KUKA KRL program: f1_Kuka_APT203T02S03.SRC

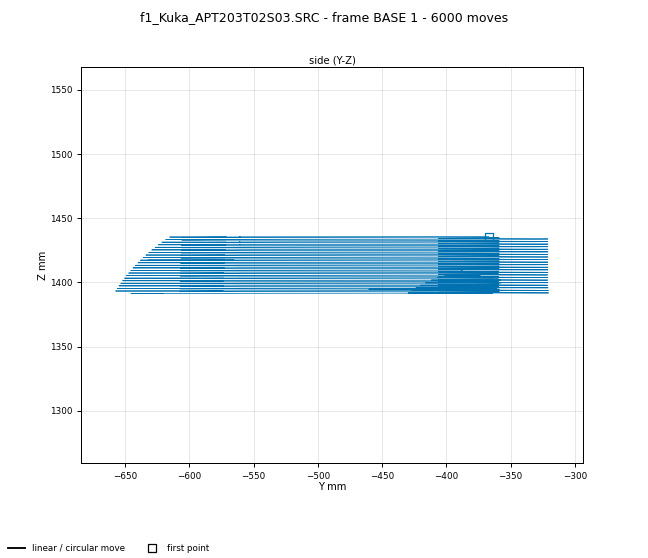
[picture p0: tool path of f1_Kuka_APT203T02S03.SRC in frame BASE 1, 6000 of 6001 moves have a stored position in this frame; points joined in program order, loops and branches not executed]
&ACCESS RVP
&REL 2
&PARAM TEMPLATE = C:\KRC\Roboter\Template\vorgabe
&PARAM EDITMASK = *
DEF f1_Kuka_APT203T02S03()


;FOLD INI;%{PE}%V3.2.0,%MKUKATPBASIS,%CINIT,%VCOMMON,%P
  ;FOLD BAS INI;%{E}%V3.2.0,%MKUKATPBASIS,%CINIT,%VINIT,%P
    GLOBAL INTERRUPT DECL 3 WHEN $STOPMESS==TRUE DO IR_STOPM ( )
    INTERRUPT ON 3
    BAS (#INITMOV,0 )
  ;ENDFOLD (BAS INI)
  ;FOLD USER INI;%{E}%V3.2.0,%MKUKATPUSER,%CINIT,%VINIT,%P
    ;Make your modifications here
  ;ENDFOLD (USER INI)
;ENDFOLD (INI)


;*** Make Null PTP Move
  PTP $pos_act

;*** Auto Load The Correct TOOL Data
  $tool=tool_data[2]

;*** Auto Load The Correct BASE Data
  $base=base_data[1]

  $ADVANCE = 5

;*** Restate Last Velocity
MMPM(30000.0)
SetRPM(8000)
LIN {X 0.139,Y -366.989,Z 1435.725,A 0.000,B 0.000,C 90.000,E1 166.408} C_DIS
LIN {X -0.133,Y -369.731,Z 1435.724,A 0.000,B 0.000,C 90.000,E1 166.284} C_DIS
LIN {X -0.049,Y -372.656,Z 1435.723,A 0.000,B 0.000,C 90.000,E1 166.061} C_DIS
LIN {X -0.133,Y -378.778,Z 1435.720,A 0.000,B 0.000,C 90.000,E1 165.574} C_DIS
LIN {X -0.061,Y -386.543,Z 1435.716,A 0.000,B 0.000,C 90.000,E1 164.866} C_DIS
LIN {X 0.126,Y -394.122,Z 1435.712,A 0.000,B 0.000,C 90.000,E1 164.102} C_DIS
LIN {X -0.061,Y -412.834,Z 1435.702,A 0.000,B 0.000,C 90.000,E1 162.417} C_DIS
LIN {X -0.188,Y -426.811,Z 1435.696,A 0.000,B 0.000,C 90.000,E1 161.221} C_DIS
LIN {X 0.041,Y -439.162,Z 1435.690,A 0.000,B 0.000,C 90.000,E1 160.134} C_DIS
LIN {X -0.042,Y -454.601,Z 1435.682,A 0.000,B 0.000,C 90.000,E1 158.847} C_DIS
LIN {X -0.244,Y -463.730,Z 1435.678,A 0.000,B 0.000,C 90.000,E1 158.103} C_DIS
LIN {X -0.043,Y -474.282,Z 1435.673,A 0.000,B 0.000,C 90.000,E1 157.177} C_DIS
LIN {X 0.193,Y -484.648,Z 1435.668,A 0.000,B 0.000,C 90.000,E1 156.230} C_DIS
LIN {X 0.112,Y -493.177,Z 1435.664,A 0.000,B 0.000,C 90.000,E1 155.433} C_DIS
LIN {X -0.238,Y -500.193,Z 1435.660,A 0.000,B 0.000,C 90.000,E1 154.793} C_DIS
LIN {X -0.084,Y -506.867,Z 1435.656,A 0.000,B 0.000,C 90.000,E1 154.076} C_DIS
LIN {X -0.024,Y -510.765,Z 1435.654,A 0.000,B 0.000,C 90.000,E1 153.640} C_DIS
LIN {X -0.152,Y -516.626,Z 1435.650,A 0.000,B 0.000,C 90.000,E1 152.922} C_DIS
LIN {X -0.204,Y -519.973,Z 1435.647,A 0.000,B 0.000,C 90.000,E1 152.487} C_DIS
LIN {X -0.159,Y -524.000,Z 1435.644,A 0.000,B 0.000,C 90.000,E1 151.897} C_DIS
LIN {X -0.081,Y -527.512,Z 1435.641,A 0.000,B 0.000,C 90.000,E1 151.307} C_DIS
LIN {X -0.125,Y -531.403,Z 1435.637,A 0.000,B 0.000,C 90.000,E1 150.589} C_DIS
LIN {X 0.009,Y -534.231,Z 1435.633,A 0.000,B 0.000,C 90.000,E1 149.999} C_DIS
LIN {X 0.019,Y -537.257,Z 1435.629,A 0.000,B 0.000,C 90.000,E1 149.282} C_DIS
LIN {X -0.271,Y -539.517,Z 1435.626,A 0.000,B 0.000,C 90.000,E1 148.742} C_DIS
LIN {X -0.078,Y -542.313,Z 1435.621,A 0.000,B 0.000,C 90.000,E1 147.867} C_DIS
LIN {X -0.041,Y -544.044,Z 1435.618,A 0.000,B 0.000,C 90.000,E1 147.296} C_DIS
LIN {X -0.062,Y -547.087,Z 1435.612,A 0.000,B 0.000,C 90.000,E1 146.167} C_DIS
LIN {X 0.115,Y -549.696,Z 1435.606,A 0.000,B 0.000,C 90.000,E1 145.022} C_DIS
LIN {X -0.096,Y -550.840,Z 1435.603,A 0.000,B 0.000,C 90.000,E1 144.482} C_DIS
LIN {X 0.145,Y -552.809,Z 1435.596,A 0.000,B 0.000,C 90.000,E1 143.336} C_DIS
LIN {X 0.346,Y -554.026,Z 1435.592,A 0.000,B 0.000,C 90.000,E1 142.477} C_DIS
LIN {X 0.271,Y -555.675,Z 1435.584,A 0.000,B 0.000,C 90.000,E1 141.090} C_DIS
LIN {X 0.141,Y -556.707,Z 1435.578,A 0.000,B 0.000,C 90.000,E1 139.989} C_DIS
LIN {X 0.039,Y -557.845,Z 1435.570,A 0.000,B 0.000,C 90.000,E1 138.609} C_DIS
LIN {X -0.041,Y -558.827,Z 1435.562,A 0.000,B 0.000,C 90.000,E1 137.229} C_DIS
LIN {X -0.185,Y -559.579,Z 1435.556,A 0.000,B 0.000,C 90.000,E1 136.134} C_DIS
LIN {X 0.071,Y -560.088,Z 1435.550,A 0.000,B 0.000,C 90.000,E1 135.000} C_DIS
LIN {X 0.002,Y -560.630,Z 1435.542,A 0.000,B 0.000,C 90.000,E1 133.623} C_DIS
LIN {X -0.035,Y -560.945,Z 1435.535,A 0.000,B 0.000,C 90.000,E1 132.243} C_DIS
LIN {X -0.060,Y -561.072,Z 1435.527,A 0.000,B 0.000,C 90.000,E1 130.862} C_DIS
LIN {X 0.097,Y -561.162,Z 1435.516,A 0.000,B 0.000,C 90.000,E1 128.910} C_DIS
LIN {X 0.142,Y -561.163,Z 1435.509,A 0.000,B 0.000,C 90.000,E1 127.523} C_DIS
LIN {X -0.055,Y -561.053,Z 1435.499,A 0.000,B 0.000,C 90.000,E1 125.884} C_DIS
LIN {X 0.103,Y -560.922,Z 1435.492,A 0.000,B 0.000,C 90.000,E1 124.485} C_DIS
LIN {X 0.254,Y -560.635,Z 1435.484,A 0.000,B 0.000,C 90.000,E1 123.086} C_DIS
LIN {X 0.083,Y -560.385,Z 1435.476,A 0.000,B 0.000,C 90.000,E1 121.720} C_DIS
LIN {X -0.090,Y -560.625,Z 1435.459,A 0.000,B 0.000,C 90.000,E1 118.693} C_DIS
LIN {X 0.023,Y -561.190,Z 1435.449,A 0.000,B 0.000,C 90.000,E1 116.744} C_DIS
LIN {X 0.086,Y -561.848,Z 1435.439,A 0.000,B 0.000,C 90.000,E1 115.079} C_DIS
LIN {X 0.115,Y -562.232,Z 1435.432,A 0.000,B 0.000,C 90.000,E1 113.695} C_DIS
LIN {X 0.247,Y -562.726,Z 1435.423,A 0.000,B 0.000,C 90.000,E1 112.025} C_DIS
LIN {X 0.174,Y -563.696,Z 1435.416,A 0.000,B 0.000,C 90.000,E1 110.791} C_DIS
LIN {X 0.095,Y -564.430,Z 1435.414,A 0.000,B 0.000,C 90.000,E1 110.482} C_DIS
LIN {X -0.307,Y -564.927,Z 1435.412,A 0.000,B 0.000,C 90.000,E1 110.248} C_DIS
LIN {X -0.215,Y -566.966,Z 1435.411,A 0.000,B 0.000,C 90.000,E1 109.939} C_DIS
LIN {X 0.217,Y -568.542,Z 1435.410,A 0.000,B 0.000,C 90.000,E1 109.758} C_DIS
LIN {X -0.209,Y -571.322,Z 1435.409,A 0.000,B 0.000,C 90.000,E1 109.577} C_DIS
LIN {X -0.175,Y -580.313,Z 1435.406,A 0.000,B 0.000,C 90.000,E1 109.014} C_DIS
LIN {X 0.231,Y -583.140,Z 1435.405,A 0.000,B 0.000,C 90.000,E1 108.779} C_DIS
LIN {X -0.178,Y -587.504,Z 1435.403,A 0.000,B 0.000,C 90.000,E1 108.489} C_DIS
LIN {X 0.008,Y -592.694,Z 1435.400,A 0.000,B 0.000,C 90.000,E1 108.000} C_DIS
LIN {X 0.320,Y -597.592,Z 1435.397,A 0.000,B 0.000,C 90.000,E1 107.457} C_DIS
LIN {X -0.290,Y -602.793,Z 1435.394,A 0.000,B 0.000,C 90.000,E1 106.858} C_DIS
LIN {X -0.042,Y -605.424,Z 1435.391,A 0.000,B 0.000,C 90.000,E1 106.441} C_DIS
LIN {X -0.313,Y -607.026,Z 1435.390,A 0.000,B 0.000,C 90.000,E1 106.205} C_DIS
LIN {X -0.042,Y -608.899,Z 1435.388,A 0.000,B 0.000,C 90.000,E1 105.788} C_DIS
LIN {X 0.194,Y -610.823,Z 1435.385,A 0.000,B 0.000,C 90.000,E1 105.245} C_DIS
LIN {X -0.060,Y -611.515,Z 1435.383,A 0.000,B 0.000,C 90.000,E1 105.009} C_DIS
LIN {X 0.034,Y -612.594,Z 1435.380,A 0.000,B 0.000,C 90.000,E1 104.481} C_DIS
LIN {X 0.042,Y -613.900,Z 1435.376,A 0.000,B 0.000,C 90.000,E1 103.703} C_DIS
LIN {X -0.086,Y -614.813,Z 1435.372,A 0.000,B 0.000,C 90.000,E1 102.939} C_DIS
LIN {X 0.033,Y -615.205,Z 1435.369,A 0.000,B 0.000,C 90.000,E1 102.411} C_DIS
LIN {X 0.156,Y -615.334,Z 1435.366,A 0.000,B 0.000,C 90.000,E1 101.883} C_DIS
LIN {X 0.158,Y -615.193,Z 1435.363,A 0.000,B 0.000,C 90.000,E1 101.366} C_DIS
LIN {X 0.283,Y -614.654,Z 1435.360,A 0.000,B 0.000,C 90.000,E1 100.838} C_DIS
LIN {X -0.202,Y -613.771,Z 1435.358,A 0.000,B 0.000,C 90.000,E1 100.366} C_DIS
LIN {X -0.197,Y -612.563,Z 1435.355,A 0.000,B 0.000,C 90.000,E1 99.849} C_DIS
LIN {X -0.095,Y -611.088,Z 1435.352,A 0.000,B 0.000,C 90.000,E1 99.321} C_DIS
LIN {X 0.252,Y -610.301,Z 1435.350,A 0.000,B 0.000,C 90.000,E1 99.029} C_DIS
LIN {X 0.239,Y -608.456,Z 1435.347,A 0.000,B 0.000,C 90.000,E1 98.511} C_DIS
LIN {X 0.123,Y -605.414,Z 1435.344,A 0.000,B 0.000,C 90.000,E1 97.871} C_DIS
LIN {X 0.016,Y -599.697,Z 1435.338,A 0.000,B 0.000,C 90.000,E1 96.834} C_DIS
LIN {X -0.252,Y -595.611,Z 1435.334,A 0.000,B 0.000,C 90.000,E1 96.201} C_DIS
LIN {X 0.231,Y -591.760,Z 1435.331,A 0.000,B 0.000,C 90.000,E1 95.625} C_DIS
LIN {X 0.011,Y -585.389,Z 1435.328,A 0.000,B 0.000,C 90.000,E1 94.992} C_DIS
LIN {X -0.058,Y -578.085,Z 1435.325,A 0.000,B 0.000,C 90.000,E1 94.416} C_DIS
LIN {X 0.163,Y -573.369,Z 1435.322,A 0.000,B 0.000,C 90.000,E1 93.955} C_DIS
LIN {X -0.164,Y -571.760,Z 1435.320,A 0.000,B 0.000,C 90.000,E1 93.669} C_DIS
LIN {X -0.139,Y -571.146,Z 1435.318,A 0.000,B 0.000,C 90.000,E1 93.326} C_DIS
LIN {X 0.212,Y -571.043,Z 1435.318,A 0.000,B 0.000,C 90.000,E1 93.154} C_DIS
LIN {X 0.110,Y -571.148,Z 1435.313,A 0.000,B 0.000,C 90.000,E1 92.350} C_DIS
LIN {X -0.222,Y -573.341,Z 1435.298,A 0.000,B 0.000,C 90.000,E1 89.656} C_DIS
LIN {X -0.082,Y -574.625,Z 1435.290,A 0.000,B 0.000,C 90.000,E1 88.282} C_DIS
LIN {X 0.272,Y -576.117,Z 1435.281,A 0.000,B 0.000,C 90.000,E1 86.617} C_DIS
LIN {X -0.248,Y -577.119,Z 1435.275,A 0.000,B 0.000,C 90.000,E1 85.584} C_DIS
LIN {X 0.219,Y -578.736,Z 1435.266,A 0.000,B 0.000,C 90.000,E1 83.913} C_DIS
LIN {X 0.154,Y -581.189,Z 1435.253,A 0.000,B 0.000,C 90.000,E1 81.489} C_DIS
LIN {X 0.060,Y -582.537,Z 1435.245,A 0.000,B 0.000,C 90.000,E1 80.151} C_DIS
LIN {X 0.141,Y -584.830,Z 1435.233,A 0.000,B 0.000,C 90.000,E1 77.993} C_DIS
LIN {X 0.221,Y -585.974,Z 1435.226,A 0.000,B 0.000,C 90.000,E1 76.645} C_DIS
LIN {X -0.109,Y -586.981,Z 1435.219,A 0.000,B 0.000,C 90.000,E1 75.338} C_DIS
LIN {X -0.098,Y -587.692,Z 1435.213,A 0.000,B 0.000,C 90.000,E1 74.267} C_DIS
LIN {X -0.158,Y -588.617,Z 1435.204,A 0.000,B 0.000,C 90.000,E1 72.670} C_DIS
LIN {X 0.139,Y -589.465,Z 1435.195,A 0.000,B 0.000,C 90.000,E1 71.040} C_DIS
LIN {X 0.101,Y -590.311,Z 1435.186,A 0.000,B 0.000,C 90.000,E1 69.444} C_DIS
LIN {X -0.020,Y -591.408,Z 1435.176,A 0.000,B 0.000,C 90.000,E1 67.592} C_DIS
LIN {X -0.027,Y -592.306,Z 1435.167,A 0.000,B 0.000,C 90.000,E1 65.997} C_DIS
LIN {X -0.274,Y -593.812,Z 1435.155,A 0.000,B 0.000,C 90.000,E1 63.896} C_DIS
LIN {X 0.065,Y -594.884,Z 1435.147,A 0.000,B 0.000,C 90.000,E1 62.538} C_DIS
LIN {X 0.275,Y -597.024,Z 1435.133,A 0.000,B 0.000,C 90.000,E1 59.871} C_DIS
LIN {X -0.248,Y -598.685,Z 1435.123,A 0.000,B 0.000,C 90.000,E1 58.074} C_DIS
LIN {X 0.263,Y -599.902,Z 1435.115,A 0.000,B 0.000,C 90.000,E1 56.707} C_DIS
LIN {X -0.047,Y -601.554,Z 1435.105,A 0.000,B 0.000,C 90.000,E1 54.895} C_DIS
LIN {X -0.219,Y -602.822,Z 1435.096,A 0.000,B 0.000,C 90.000,E1 53.336} C_DIS
LIN {X 0.215,Y -603.813,Z 1435.089,A 0.000,B 0.000,C 90.000,E1 51.984} C_DIS
LIN {X -0.030,Y -604.760,Z 1435.080,A 0.000,B 0.000,C 90.000,E1 50.436} C_DIS
LIN {X -0.183,Y -605.178,Z 1435.076,A 0.000,B 0.000,C 90.000,E1 49.666} C_DIS
LIN {X 0.188,Y -605.443,Z 1435.069,A 0.000,B 0.000,C 90.000,E1 48.324} C_DIS
LIN {X -0.292,Y -605.672,Z 1435.058,A 0.000,B 0.000,C 90.000,E1 46.539} C_DIS
LIN {X 0.030,Y -605.750,Z 1435.051,A 0.000,B 0.000,C 90.000,E1 45.202} C_DIS
LIN {X -0.313,Y -605.439,Z 1435.045,A 0.000,B 0.000,C 90.000,E1 44.190} C_DIS
LIN {X 0.010,Y -604.840,Z 1435.038,A 0.000,B 0.000,C 90.000,E1 42.852} C_DIS
LIN {X -0.085,Y -603.901,Z 1435.031,A 0.000,B 0.000,C 90.000,E1 41.553} C_DIS
LIN {X -0.238,Y -603.180,Z 1435.026,A 0.000,B 0.000,C 90.000,E1 40.782} C_DIS
LIN {X 0.098,Y -601.757,Z 1435.019,A 0.000,B 0.000,C 90.000,E1 39.439} C_DIS
LIN {X 0.157,Y -600.481,Z 1435.013,A 0.000,B 0.000,C 90.000,E1 38.382} C_DIS
LIN {X 0.058,Y -598.543,Z 1435.006,A 0.000,B 0.000,C 90.000,E1 37.076} C_DIS
LIN {X 0.052,Y -596.081,Z 1434.999,A 0.000,B 0.000,C 90.000,E1 35.758} C_DIS
LIN {X -0.136,Y -593.171,Z 1434.991,A 0.000,B 0.000,C 90.000,E1 34.452} C_DIS
LIN {X 0.170,Y -591.220,Z 1434.987,A 0.000,B 0.000,C 90.000,E1 33.627} C_DIS
LIN {X 0.332,Y -588.313,Z 1434.981,A 0.000,B 0.000,C 90.000,E1 32.546} C_DIS
LIN {X -0.097,Y -586.776,Z 1434.978,A 0.000,B 0.000,C 90.000,E1 32.054} C_DIS
LIN {X -0.171,Y -584.094,Z 1434.974,A 0.000,B 0.000,C 90.000,E1 31.258} C_DIS
LIN {X -0.133,Y -582.079,Z 1434.971,A 0.000,B 0.000,C 90.000,E1 30.718} C_DIS
LIN {X -0.112,Y -579.882,Z 1434.968,A 0.000,B 0.000,C 90.000,E1 30.178} C_DIS
LIN {X 0.246,Y -576.285,Z 1434.963,A 0.000,B 0.000,C 90.000,E1 29.333} C_DIS
LIN {X -0.138,Y -572.981,Z 1434.959,A 0.000,B 0.000,C 90.000,E1 28.693} C_DIS
LIN {X 0.146,Y -568.644,Z 1434.955,A 0.000,B 0.000,C 90.000,E1 27.847} C_DIS
LIN {X 0.283,Y -563.075,Z 1434.949,A 0.000,B 0.000,C 90.000,E1 26.873} C_DIS
LIN {X -0.005,Y -556.116,Z 1434.943,A 0.000,B 0.000,C 90.000,E1 25.796} C_DIS
LIN {X 0.079,Y -550.567,Z 1434.939,A 0.000,B 0.000,C 90.000,E1 24.951} C_DIS
LIN {X 0.109,Y -546.505,Z 1434.936,A 0.000,B 0.000,C 90.000,E1 24.387} C_DIS
LIN {X -0.019,Y -540.965,Z 1434.932,A 0.000,B 0.000,C 90.000,E1 23.695} C_DIS
LIN {X 0.300,Y -535.092,Z 1434.928,A 0.000,B 0.000,C 90.000,E1 22.950} C_DIS
LIN {X -0.249,Y -527.574,Z 1434.923,A 0.000,B 0.000,C 90.000,E1 22.153} C_DIS
LIN {X -0.192,Y -518.481,Z 1434.917,A 0.000,B 0.000,C 90.000,E1 21.153} C_DIS
LIN {X -0.220,Y -512.109,Z 1434.914,A 0.000,B 0.000,C 90.000,E1 20.482} C_DIS
LIN {X 0.092,Y -501.330,Z 1434.907,A 0.000,B 0.000,C 90.000,E1 19.322} C_DIS
LIN {X -0.015,Y -487.754,Z 1434.900,A 0.000,B 0.000,C 90.000,E1 17.946} C_DIS
LIN {X -0.074,Y -470.249,Z 1434.889,A 0.000,B 0.000,C 90.000,E1 16.079} C_DIS
LIN {X -0.198,Y -452.851,Z 1434.878,A 0.000,B 0.000,C 90.000,E1 14.120} C_DIS
LIN {X 0.206,Y -444.598,Z 1434.873,A 0.000,B 0.000,C 90.000,E1 13.119} C_DIS
LIN {X -0.161,Y -440.352,Z 1434.870,A 0.000,B 0.000,C 90.000,E1 12.703} C_DIS
LIN {X -0.110,Y -435.815,Z 1434.868,A 0.000,B 0.000,C 90.000,E1 12.243} C_DIS
LIN {X -0.151,Y -431.034,Z 1434.866,A 0.000,B 0.000,C 90.000,E1 11.827} C_DIS
LIN {X 0.079,Y -427.565,Z 1434.864,A 0.000,B 0.000,C 90.000,E1 11.535} C_DIS
LIN {X 0.097,Y -423.730,Z 1434.863,A 0.000,B 0.000,C 90.000,E1 11.299} C_DIS
LIN {X 0.019,Y -420.614,Z 1434.862,A 0.000,B 0.000,C 90.000,E1 11.186} C_DIS
LIN {X -0.096,Y -419.777,Z 1434.862,A 0.000,B 0.000,C 90.000,E1 11.186} C_DIS
LIN {X -0.117,Y -367.196,Z 1434.862,A 0.000,B 0.000,C 90.000,E1 11.186} C_DIS
LIN {X -0.112,Y -366.497,Z 1434.855,A 0.000,B 0.000,C 90.000,E1 9.962} C_DIS
LIN {X 0.185,Y -361.797,Z 1434.822,A 0.000,B 0.000,C 90.000,E1 3.955} C_DIS
LIN {X 0.070,Y -360.903,Z 1434.801,A 0.000,B 0.000,C 90.000,E1 0.229} C_DIS
LIN {X -0.053,Y -359.426,Z 1434.770,A 0.000,B 0.000,C 90.000,E1 354.546} C_DIS
LIN {X 0.070,Y -358.890,Z 1434.759,A 0.000,B 0.000,C 90.000,E1 352.648} C_DIS
LIN {X -0.020,Y -359.563,Z 1434.726,A 0.000,B 0.000,C 90.000,E1 346.645} C_DIS
LIN {X 0.001,Y -361.801,Z 1434.684,A 0.000,B 0.000,C 90.000,E1 339.135} C_DIS
LIN {X -0.154,Y -362.053,Z 1434.680,A 0.000,B 0.000,C 90.000,E1 338.411} C_DIS
LIN {X 0.189,Y -365.980,Z 1434.643,A 0.000,B 0.000,C 90.000,E1 331.641} C_DIS
LIN {X 0.029,Y -366.387,Z 1434.639,A 0.000,B 0.000,C 90.000,E1 330.923} C_DIS
LIN {X -0.031,Y -371.355,Z 1434.604,A 0.000,B 0.000,C 90.000,E1 324.642} C_DIS
LIN {X -0.043,Y -371.766,Z 1434.602,A 0.000,B 0.000,C 90.000,E1 324.276} C_DIS
LIN {X 0.013,Y -377.358,Z 1434.567,A 0.000,B 0.000,C 90.000,E1 318.038} C_DIS
LIN {X 0.012,Y -378.235,Z 1434.563,A 0.000,B 0.000,C 90.000,E1 317.310} C_DIS
LIN {X 0.002,Y -383.940,Z 1434.531,A 0.000,B 0.000,C 90.000,E1 311.515} C_DIS
LIN {X 0.088,Y -384.893,Z 1434.527,A 0.000,B 0.000,C 90.000,E1 310.782} C_DIS
LIN {X 0.262,Y -390.610,Z 1434.495,A 0.000,B 0.000,C 90.000,E1 305.025} C_DIS
LIN {X 0.106,Y -391.104,Z 1434.493,A 0.000,B 0.000,C 90.000,E1 304.692} C_DIS
LIN {X 0.022,Y -391.648,Z 1434.489,A 0.000,B 0.000,C 90.000,E1 303.992} C_DIS
LIN {X -0.080,Y -396.825,Z 1434.459,A 0.000,B 0.000,C 90.000,E1 298.693} C_DIS
LIN {X -0.210,Y -397.120,Z 1434.457,A 0.000,B 0.000,C 90.000,E1 298.359} C_DIS
LIN {X -0.055,Y -401.597,Z 1434.426,A 0.000,B 0.000,C 90.000,E1 292.717} C_DIS
LIN {X 0.222,Y -404.659,Z 1434.395,A 0.000,B 0.000,C 90.000,E1 287.094} C_DIS
LIN {X -0.079,Y -404.735,Z 1434.391,A 0.000,B 0.000,C 90.000,E1 286.441} C_DIS
LIN {X 0.214,Y -406.099,Z 1434.364,A 0.000,B 0.000,C 90.000,E1 281.535} C_DIS
LIN {X -0.176,Y -406.094,Z 1434.362,A 0.000,B 0.000,C 90.000,E1 281.243} C_DIS
LIN {X -0.097,Y -405.680,Z 1434.333,A 0.000,B 0.000,C 90.000,E1 276.024} C_DIS
LIN {X -0.165,Y -405.058,Z 1434.328,A 0.000,B 0.000,C 90.000,E1 274.992} C_DIS
LIN {X -0.060,Y -403.497,Z 1434.304,A 0.000,B 0.000,C 90.000,E1 270.802} C_DIS
LIN {X -0.092,Y -403.288,Z 1434.302,A 0.000,B 0.000,C 90.000,E1 270.458} C_DIS
LIN {X 0.091,Y -398.931,Z 1434.271,A 0.000,B 0.000,C 90.000,E1 264.837} C_DIS
LIN {X -0.040,Y -393.108,Z 1434.242,A 0.000,B 0.000,C 90.000,E1 259.567} C_DIS
LIN {X -0.079,Y -392.835,Z 1434.240,A 0.000,B 0.000,C 90.000,E1 259.218} C_DIS
LIN {X 0.034,Y -385.993,Z 1434.212,A 0.000,B 0.000,C 90.000,E1 254.212} C_DIS
LIN {X -0.026,Y -385.267,Z 1434.208,A 0.000,B 0.000,C 90.000,E1 253.504} C_DIS
LIN {X -0.004,Y -384.768,Z 1434.206,A 0.000,B 0.000,C 90.000,E1 253.142} C_DIS
LIN {X 0.221,Y -377.973,Z 1434.182,A 0.000,B 0.000,C 90.000,E1 248.773} C_DIS
LIN {X -0.044,Y -376.233,Z 1434.174,A 0.000,B 0.000,C 90.000,E1 247.358} C_DIS
LIN {X 0.057,Y -374.944,Z 1434.170,A 0.000,B 0.000,C 90.000,E1 246.613} C_DIS
LIN {X -0.208,Y -368.417,Z 1434.148,A 0.000,B 0.000,C 90.000,E1 242.615} C_DIS
LIN {X 0.097,Y -366.047,Z 1434.137,A 0.000,B 0.000,C 90.000,E1 240.717} C_DIS
LIN {X 0.004,Y -359.196,Z 1434.115,A 0.000,B 0.000,C 90.000,E1 236.628} C_DIS
LIN {X 0.021,Y -355.842,Z 1434.100,A 0.000,B 0.000,C 90.000,E1 233.989} C_DIS
LIN {X -0.173,Y -348.793,Z 1434.075,A 0.000,B 0.000,C 90.000,E1 229.461} C_DIS
LIN {X -0.097,Y -346.185,Z 1434.062,A 0.000,B 0.000,C 90.000,E1 227.148} C_DIS
LIN {X -0.088,Y -345.065,Z 1434.058,A 0.000,B 0.000,C 90.000,E1 226.377} C_DIS
LIN {X 0.094,Y -338.586,Z 1434.030,A 0.000,B 0.000,C 90.000,E1 221.310} C_DIS
LIN {X 0.094,Y -336.840,Z 1434.019,A 0.000,B 0.000,C 90.000,E1 219.358} C_DIS
LIN {X 0.014,Y -330.861,Z 1433.988,A 0.000,B 0.000,C 90.000,E1 213.865} C_DIS
LIN {X 0.149,Y -329.296,Z 1433.975,A 0.000,B 0.000,C 90.000,E1 211.465} C_DIS
LIN {X -0.154,Y -324.669,Z 1433.942,A 0.000,B 0.000,C 90.000,E1 205.540} C_DIS
LIN {X 0.174,Y -323.837,Z 1433.928,A 0.000,B 0.000,C 90.000,E1 203.078} C_DIS
LIN {X -0.017,Y -321.124,Z 1433.881,A 0.000,B 0.000,C 90.000,E1 194.662} C_DIS
LIN {X 0.138,Y -320.932,Z 1433.877,A 0.000,B 0.000,C 90.000,E1 193.828} C_DIS
LIN {X -0.076,Y -321.562,Z 1433.832,A 0.000,B 0.000,C 90.000,E1 185.796} C_DIS
LIN {X -0.143,Y -324.415,Z 1433.790,A 0.000,B 0.000,C 90.000,E1 178.165} C_DIS
LIN {X -0.141,Y -325.376,Z 1433.783,A 0.000,B 0.000,C 90.000,E1 176.963} C_DIS
LIN {X -0.100,Y -329.112,Z 1433.750,A 0.000,B 0.000,C 90.000,E1 170.971} C_DIS
LIN {X 0.124,Y -333.112,Z 1433.730,A 0.000,B 0.000,C 90.000,E1 167.409} C_DIS
LIN {X 0.112,Y -355.729,Z 1433.730,A 0.000,B 0.000,C 90.000,E1 167.409} C_DIS
LIN {X -0.132,Y -357.447,Z 1433.730,A 0.000,B 0.000,C 90.000,E1 167.409} C_DIS
LIN {X 0.008,Y -359.821,Z 1433.729,A 0.000,B 0.000,C 90.000,E1 167.285} C_DIS
LIN {X 0.102,Y -362.424,Z 1433.729,A 0.000,B 0.000,C 90.000,E1 167.117} C_DIS
LIN {X -0.043,Y -365.285,Z 1433.727,A 0.000,B 0.000,C 90.000,E1 166.937} C_DIS
LIN {X -0.188,Y -369.813,Z 1433.725,A 0.000,B 0.000,C 90.000,E1 166.589} C_DIS
LIN {X 0.026,Y -375.870,Z 1433.722,A 0.000,B 0.000,C 90.000,E1 165.992} C_DIS
LIN {X 0.077,Y -383.469,Z 1433.718,A 0.000,B 0.000,C 90.000,E1 165.227} C_DIS
LIN {X -0.010,Y -397.106,Z 1433.710,A 0.000,B 0.000,C 90.000,E1 163.866} C_DIS
LIN {X 0.091,Y -414.197,Z 1433.702,A 0.000,B 0.000,C 90.000,E1 162.308} C_DIS
LIN {X 0.208,Y -428.111,Z 1433.695,A 0.000,B 0.000,C 90.000,E1 161.094} C_DIS
LIN {X 0.028,Y -442.117,Z 1433.689,A 0.000,B 0.000,C 90.000,E1 159.934} C_DIS
LIN {X 0.121,Y -457.244,Z 1433.682,A 0.000,B 0.000,C 90.000,E1 158.646} C_DIS
LIN {X -0.188,Y -469.309,Z 1433.676,A 0.000,B 0.000,C 90.000,E1 157.667} C_DIS
LIN {X -0.059,Y -479.763,Z 1433.671,A 0.000,B 0.000,C 90.000,E1 156.741} C_DIS
LIN {X -0.186,Y -486.922,Z 1433.667,A 0.000,B 0.000,C 90.000,E1 156.102} C_DIS
LIN {X -0.083,Y -496.799,Z 1433.662,A 0.000,B 0.000,C 90.000,E1 155.153} C_DIS
LIN {X 0.061,Y -503.454,Z 1433.658,A 0.000,B 0.000,C 90.000,E1 154.460} C_DIS
LIN {X 0.172,Y -507.445,Z 1433.656,A 0.000,B 0.000,C 90.000,E1 154.024} C_DIS
LIN {X -0.231,Y -511.337,Z 1433.653,A 0.000,B 0.000,C 90.000,E1 153.640} C_DIS
LIN {X 0.087,Y -517.167,Z 1433.649,A 0.000,B 0.000,C 90.000,E1 152.871} C_DIS
LIN {X 0.037,Y -520.484,Z 1433.647,A 0.000,B 0.000,C 90.000,E1 152.436} C_DIS
LIN {X 0.086,Y -524.476,Z 1433.644,A 0.000,B 0.000,C 90.000,E1 151.847} C_DIS
LIN {X 0.167,Y -527.972,Z 1433.641,A 0.000,B 0.000,C 90.000,E1 151.257} C_DIS
LIN {X 0.125,Y -531.869,Z 1433.636,A 0.000,B 0.000,C 90.000,E1 150.539} C_DIS
LIN {X -0.202,Y -534.631,Z 1433.633,A 0.000,B 0.000,C 90.000,E1 149.999} C_DIS
LIN {X -0.189,Y -537.680,Z 1433.629,A 0.000,B 0.000,C 90.000,E1 149.282} C_DIS
LIN {X 0.264,Y -539.878,Z 1433.626,A 0.000,B 0.000,C 90.000,E1 148.663} C_DIS
LIN {X -0.006,Y -541.789,Z 1433.623,A 0.000,B 0.000,C 90.000,E1 148.122} C_DIS
LIN {X 0.216,Y -544.348,Z 1433.618,A 0.000,B 0.000,C 90.000,E1 147.248} C_DIS
LIN {X 0.008,Y -546.662,Z 1433.614,A 0.000,B 0.000,C 90.000,E1 146.421} C_DIS
LIN {X -0.176,Y -548.681,Z 1433.609,A 0.000,B 0.000,C 90.000,E1 145.595} C_DIS
LIN {X -0.025,Y -550.545,Z 1433.604,A 0.000,B 0.000,C 90.000,E1 144.736} C_DIS
LIN {X -0.171,Y -552.091,Z 1433.599,A 0.000,B 0.000,C 90.000,E1 143.909} C_DIS
LIN {X 0.022,Y -553.382,Z 1433.595,A 0.000,B 0.000,C 90.000,E1 143.050} C_DIS
LIN {X 0.228,Y -554.491,Z 1433.590,A 0.000,B 0.000,C 90.000,E1 142.190} C_DIS
LIN {X 0.085,Y -555.779,Z 1433.584,A 0.000,B 0.000,C 90.000,E1 141.090} C_DIS
LIN {X -0.044,Y -556.801,Z 1433.578,A 0.000,B 0.000,C 90.000,E1 139.989} C_DIS
LIN {X -0.145,Y -557.909,Z 1433.570,A 0.000,B 0.000,C 90.000,E1 138.609} C_DIS
LIN {X -0.224,Y -558.869,Z 1433.562,A 0.000,B 0.000,C 90.000,E1 137.229} C_DIS
LIN {X -0.368,Y -559.594,Z 1433.556,A 0.000,B 0.000,C 90.000,E1 136.134} C_DIS
LIN {X -0.112,Y -560.099,Z 1433.550,A 0.000,B 0.000,C 90.000,E1 135.000} C_DIS
LIN {X -0.181,Y -560.619,Z 1433.542,A 0.000,B 0.000,C 90.000,E1 133.623} C_DIS
LIN {X 0.159,Y -560.924,Z 1433.535,A 0.000,B 0.000,C 90.000,E1 132.204} C_DIS
LIN {X 0.122,Y -561.038,Z 1433.527,A 0.000,B 0.000,C 90.000,E1 130.825} C_DIS
LIN {X -0.182,Y -561.136,Z 1433.518,A 0.000,B 0.000,C 90.000,E1 129.197} C_DIS
LIN {X -0.140,Y -561.152,Z 1433.510,A 0.000,B 0.000,C 90.000,E1 127.810} C_DIS
LIN {X -0.008,Y -561.070,Z 1433.501,A 0.000,B 0.000,C 90.000,E1 126.137} C_DIS
LIN {X -0.082,Y -560.919,Z 1433.492,A 0.000,B 0.000,C 90.000,E1 124.485} C_DIS
LIN {X 0.069,Y -560.653,Z 1433.484,A 0.000,B 0.000,C 90.000,E1 123.086} C_DIS
LIN {X 0.165,Y -560.344,Z 1433.475,A 0.000,B 0.000,C 90.000,E1 121.416} C_DIS
LIN {X 0.283,Y -560.695,Z 1433.458,A 0.000,B 0.000,C 90.000,E1 118.359} C_DIS
LIN {X -0.161,Y -561.224,Z 1433.448,A 0.000,B 0.000,C 90.000,E1 116.744} C_DIS
LIN {X -0.098,Y -561.881,Z 1433.439,A 0.000,B 0.000,C 90.000,E1 115.079} C_DIS
LIN {X -0.069,Y -562.245,Z 1433.432,A 0.000,B 0.000,C 90.000,E1 113.695} C_DIS
LIN {X 0.064,Y -562.832,Z 1433.422,A 0.000,B 0.000,C 90.000,E1 112.025} C_DIS
LIN {X 0.181,Y -563.466,Z 1433.419,A 0.000,B 0.000,C 90.000,E1 111.461} C_DIS
LIN {X 0.095,Y -563.971,Z 1433.416,A 0.000,B 0.000,C 90.000,E1 110.918} C_DIS
LIN {X -0.070,Y -565.058,Z 1433.414,A 0.000,B 0.000,C 90.000,E1 110.556} C_DIS
LIN {X -0.081,Y -567.521,Z 1433.412,A 0.000,B 0.000,C 90.000,E1 110.248} C_DIS
LIN {X -0.182,Y -569.009,Z 1433.412,A 0.000,B 0.000,C 90.000,E1 110.120} C_DIS
LIN {X 0.045,Y -575.620,Z 1433.409,A 0.000,B 0.000,C 90.000,E1 109.685} C_DIS
LIN {X 0.022,Y -583.296,Z 1433.407,A 0.000,B 0.000,C 90.000,E1 109.214} C_DIS
LIN {X 0.213,Y -588.749,Z 1433.405,A 0.000,B 0.000,C 90.000,E1 108.779} C_DIS
LIN {X -0.302,Y -593.935,Z 1433.402,A 0.000,B 0.000,C 90.000,E1 108.362} C_DIS
LIN {X 0.146,Y -597.660,Z 1433.400,A 0.000,B 0.000,C 90.000,E1 107.946} C_DIS
LIN {X 0.090,Y -599.952,Z 1433.398,A 0.000,B 0.000,C 90.000,E1 107.692} C_DIS
LIN {X 0.325,Y -603.290,Z 1433.396,A 0.000,B 0.000,C 90.000,E1 107.275} C_DIS
LIN {X -0.274,Y -607.958,Z 1433.393,A 0.000,B 0.000,C 90.000,E1 106.677} C_DIS
LIN {X 0.262,Y -608.806,Z 1433.392,A 0.000,B 0.000,C 90.000,E1 106.496} C_DIS
LIN {X 0.083,Y -612.706,Z 1433.387,A 0.000,B 0.000,C 90.000,E1 105.733} C_DIS
LIN {X 0.106,Y -614.852,Z 1433.383,A 0.000,B 0.000,C 90.000,E1 104.954} C_DIS
LIN {X 0.224,Y -615.951,Z 1433.380,A 0.000,B 0.000,C 90.000,E1 104.426} C_DIS
LIN {X -0.195,Y -617.867,Z 1433.373,A 0.000,B 0.000,C 90.000,E1 103.175} C_DIS
LIN {X -0.054,Y -618.290,Z 1433.370,A 0.000,B 0.000,C 90.000,E1 102.647} C_DIS
LIN {X -0.139,Y -618.364,Z 1433.366,A 0.000,B 0.000,C 90.000,E1 101.883} C_DIS
LIN {X -0.117,Y -618.179,Z 1433.363,A 0.000,B 0.000,C 90.000,E1 101.366} C_DIS
LIN {X 0.030,Y -617.684,Z 1433.360,A 0.000,B 0.000,C 90.000,E1 100.838} C_DIS
LIN {X -0.068,Y -616.225,Z 1433.356,A 0.000,B 0.000,C 90.000,E1 100.074} C_DIS
LIN {X -0.045,Y -614.909,Z 1433.353,A 0.000,B 0.000,C 90.000,E1 99.557} C_DIS
LIN {X 0.071,Y -613.339,Z 1433.350,A 0.000,B 0.000,C 90.000,E1 99.029} C_DIS
LIN {X 0.079,Y -611.517,Z 1433.347,A 0.000,B 0.000,C 90.000,E1 98.511} C_DIS
LIN {X -0.012,Y -608.737,Z 1433.344,A 0.000,B 0.000,C 90.000,E1 97.871} C_DIS
LIN {X -0.073,Y -602.983,Z 1433.338,A 0.000,B 0.000,C 90.000,E1 96.834} C_DIS
LIN {X 0.282,Y -599.196,Z 1433.334,A 0.000,B 0.000,C 90.000,E1 96.144} C_DIS
LIN {X 0.198,Y -595.406,Z 1433.331,A 0.000,B 0.000,C 90.000,E1 95.625} C_DIS
LIN {X 0.278,Y -592.038,Z 1433.329,A 0.000,B 0.000,C 90.000,E1 95.220} C_DIS
LIN {X -0.087,Y -589.468,Z 1433.328,A 0.000,B 0.000,C 90.000,E1 94.992} C_DIS
LIN {X 0.211,Y -583.761,Z 1433.325,A 0.000,B 0.000,C 90.000,E1 94.473} C_DIS
LIN {X -0.257,Y -577.847,Z 1433.323,A 0.000,B 0.000,C 90.000,E1 94.069} C_DIS
LIN {X 0.175,Y -573.963,Z 1433.321,A 0.000,B 0.000,C 90.000,E1 93.669} C_DIS
LIN {X 0.004,Y -572.411,Z 1433.319,A 0.000,B 0.000,C 90.000,E1 93.440} C_DIS
LIN {X -0.105,Y -572.025,Z 1433.319,A 0.000,B 0.000,C 90.000,E1 93.383} C_DIS
LIN {X 0.142,Y -571.475,Z 1433.318,A 0.000,B 0.000,C 90.000,E1 93.154} C_DIS
LIN {X 0.107,Y -571.475,Z 1433.315,A 0.000,B 0.000,C 90.000,E1 92.751} C_DIS
LIN {X 0.021,Y -571.213,Z 1433.313,A 0.000,B 0.000,C 90.000,E1 92.350} C_DIS
LIN {X 0.263,Y -573.455,Z 1433.297,A 0.000,B 0.000,C 90.000,E1 89.484} C_DIS
LIN {X -0.151,Y -574.728,Z 1433.290,A 0.000,B 0.000,C 90.000,E1 88.165} C_DIS
LIN {X 0.187,Y -576.235,Z 1433.281,A 0.000,B 0.000,C 90.000,E1 86.502} C_DIS
LIN {X 0.241,Y -577.250,Z 1433.275,A 0.000,B 0.000,C 90.000,E1 85.412} C_DIS
LIN {X 0.132,Y -578.859,Z 1433.266,A 0.000,B 0.000,C 90.000,E1 83.799} C_DIS
LIN {X 0.277,Y -580.774,Z 1433.255,A 0.000,B 0.000,C 90.000,E1 81.894} C_DIS
LIN {X -0.054,Y -581.918,Z 1433.249,A 0.000,B 0.000,C 90.000,E1 80.849} C_DIS
LIN {X 0.105,Y -583.559,Z 1433.240,A 0.000,B 0.000,C 90.000,E1 79.218} C_DIS
LIN {X 0.047,Y -585.013,Z 1433.233,A 0.000,B 0.000,C 90.000,E1 77.881} C_DIS
LIN {X -0.061,Y -586.338,Z 1433.224,A 0.000,B 0.000,C 90.000,E1 76.284} C_DIS
LIN {X -0.210,Y -587.119,Z 1433.218,A 0.000,B 0.000,C 90.000,E1 75.227} C_DIS
LIN {X -0.203,Y -587.831,Z 1433.212,A 0.000,B 0.000,C 90.000,E1 74.157} C_DIS
LIN {X -0.094,Y -588.736,Z 1433.203,A 0.000,B 0.000,C 90.000,E1 72.543} C_DIS
LIN {X 0.211,Y -589.565,Z 1433.194,A 0.000,B 0.000,C 90.000,E1 70.913} C_DIS
LIN {X 0.299,Y -590.305,Z 1433.187,A 0.000,B 0.000,C 90.000,E1 69.571} C_DIS
LIN {X 0.283,Y -591.196,Z 1433.178,A 0.000,B 0.000,C 90.000,E1 67.975} C_DIS
LIN {X -0.375,Y -592.349,Z 1433.167,A 0.000,B 0.000,C 90.000,E1 66.177} C_DIS
LIN {X -0.083,Y -593.772,Z 1433.156,A 0.000,B 0.000,C 90.000,E1 64.024} C_DIS
LIN {X 0.166,Y -595.042,Z 1433.147,A 0.000,B 0.000,C 90.000,E1 62.410} C_DIS
LIN {X -0.048,Y -596.991,Z 1433.134,A 0.000,B 0.000,C 90.000,E1 60.049} C_DIS
LIN {X 0.039,Y -598.402,Z 1433.125,A 0.000,B 0.000,C 90.000,E1 58.456} C_DIS
LIN {X 0.227,Y -599.624,Z 1433.118,A 0.000,B 0.000,C 90.000,E1 57.120} C_DIS
LIN {X 0.162,Y -601.034,Z 1433.109,A 0.000,B 0.000,C 90.000,E1 55.548} C_DIS
LIN {X -0.280,Y -602.185,Z 1433.101,A 0.000,B 0.000,C 90.000,E1 54.276} C_DIS
LIN {X 0.142,Y -603.234,Z 1433.094,A 0.000,B 0.000,C 90.000,E1 52.924} C_DIS
LIN {X -0.157,Y -603.968,Z 1433.088,A 0.000,B 0.000,C 90.000,E1 51.904} C_DIS
LIN {X 0.069,Y -604.953,Z 1433.080,A 0.000,B 0.000,C 90.000,E1 50.312} C_DIS
LIN {X -0.084,Y -605.350,Z 1433.075,A 0.000,B 0.000,C 90.000,E1 49.542} C_DIS
LIN {X -0.171,Y -605.572,Z 1433.068,A 0.000,B 0.000,C 90.000,E1 48.243} C_DIS
LIN {X -0.037,Y -605.795,Z 1433.059,A 0.000,B 0.000,C 90.000,E1 46.662} C_DIS
LIN {X 0.105,Y -605.858,Z 1433.051,A 0.000,B 0.000,C 90.000,E1 45.081} C_DIS
LIN {X 0.193,Y -605.513,Z 1433.045,A 0.000,B 0.000,C 90.000,E1 44.028} C_DIS
LIN {X 0.050,Y -605.206,Z 1433.040,A 0.000,B 0.000,C 90.000,E1 43.257} C_DIS
LIN {X 0.120,Y -604.545,Z 1433.035,A 0.000,B 0.000,C 90.000,E1 42.204} C_DIS
LIN {X 0.218,Y -603.763,Z 1433.029,A 0.000,B 0.000,C 90.000,E1 41.148} C_DIS
LIN {X 0.308,Y -602.691,Z 1433.023,A 0.000,B 0.000,C 90.000,E1 40.092} C_DIS
LIN {X -0.218,Y -601.204,Z 1433.016,A 0.000,B 0.000,C 90.000,E1 38.830} C_DIS
LIN {X -0.055,Y -598.970,Z 1433.007,A 0.000,B 0.000,C 90.000,E1 37.237} C_DIS
LIN {X 0.067,Y -597.069,Z 1433.001,A 0.000,B 0.000,C 90.000,E1 36.171} C_DIS
LIN {X -0.067,Y -595.514,Z 1432.997,A 0.000,B 0.000,C 90.000,E1 35.391} C_DIS
LIN {X 0.001,Y -593.152,Z 1432.991,A 0.000,B 0.000,C 90.000,E1 34.326} C_DIS
LIN {X 0.310,Y -591.199,Z 1432.986,A 0.000,B 0.000,C 90.000,E1 33.499} C_DIS
LIN {X -0.022,Y -588.287,Z 1432.980,A 0.000,B 0.000,C 90.000,E1 32.467} C_DIS
LIN {X 0.044,Y -586.716,Z 1432.977,A 0.000,B 0.000,C 90.000,E1 31.926} C_DIS
LIN {X -0.029,Y -583.943,Z 1432.973,A 0.000,B 0.000,C 90.000,E1 31.131} C_DIS
LIN {X 0.008,Y -581.897,Z 1432.970,A 0.000,B 0.000,C 90.000,E1 30.590} C_DIS
LIN {X -0.112,Y -578.510,Z 1432.965,A 0.000,B 0.000,C 90.000,E1 29.795} C_DIS
LIN {X 0.236,Y -574.818,Z 1432.961,A 0.000,B 0.000,C 90.000,E1 28.949} C_DIS
LIN {X 0.113,Y -571.347,Z 1432.957,A 0.000,B 0.000,C 90.000,E1 28.281} C_DIS
LIN {X -0.221,Y -568.360,Z 1432.954,A 0.000,B 0.000,C 90.000,E1 27.769} C_DIS
LIN {X -0.087,Y -562.823,Z 1432.949,A 0.000,B 0.000,C 90.000,E1 26.796} C_DIS
LIN {X 0.122,Y -555.808,Z 1432.943,A 0.000,B 0.000,C 90.000,E1 25.668} C_DIS
LIN {X -0.032,Y -550.167,Z 1432.938,A 0.000,B 0.000,C 90.000,E1 24.847} C_DIS
LIN {X 0.225,Y -546.095,Z 1432.935,A 0.000,B 0.000,C 90.000,E1 24.259} C_DIS
LIN {X 0.223,Y -541.680,Z 1432.932,A 0.000,B 0.000,C 90.000,E1 23.695} C_DIS
LIN {X -0.296,Y -534.602,Z 1432.927,A 0.000,B 0.000,C 90.000,E1 22.898} C_DIS
LIN {X -0.127,Y -527.110,Z 1432.922,A 0.000,B 0.000,C 90.000,E1 22.025} C_DIS
LIN {X -0.066,Y -516.994,Z 1432.916,A 0.000,B 0.000,C 90.000,E1 20.918} C_DIS
LIN {X -0.123,Y -506.356,Z 1432.910,A 0.000,B 0.000,C 90.000,E1 19.812} C_DIS
LIN {X -0.125,Y -496.857,Z 1432.905,A 0.000,B 0.000,C 90.000,E1 18.833} C_DIS
LIN {X 0.029,Y -479.211,Z 1432.894,A 0.000,B 0.000,C 90.000,E1 16.985} C_DIS
LIN {X 0.069,Y -464.503,Z 1432.885,A 0.000,B 0.000,C 90.000,E1 15.371} C_DIS
LIN {X 0.018,Y -449.893,Z 1432.876,A 0.000,B 0.000,C 90.000,E1 13.703} C_DIS
LIN {X -0.095,Y -439.325,Z 1432.869,A 0.000,B 0.000,C 90.000,E1 12.479} C_DIS
LIN {X 0.080,Y -433.526,Z 1432.866,A 0.000,B 0.000,C 90.000,E1 11.827} C_DIS
LIN {X 0.183,Y -428.878,Z 1432.863,A 0.000,B 0.000,C 90.000,E1 11.366} C_DIS
LIN {X 0.165,Y -423.970,Z 1432.861,A 0.000,B 0.000,C 90.000,E1 10.950} C_DIS
LIN {X 0.009,Y -420.455,Z 1432.860,A 0.000,B 0.000,C 90.000,E1 10.715} C_DIS
LIN {X -0.008,Y -418.605,Z 1432.859,A 0.000,B 0.000,C 90.000,E1 10.602} C_DIS
LIN {X -0.024,Y -416.278,Z 1432.858,A 0.000,B 0.000,C 90.000,E1 10.489} C_DIS
LIN {X -0.071,Y -414.076,Z 1432.858,A 0.000,B 0.000,C 90.000,E1 10.433} C_DIS
LIN {X -0.033,Y -413.508,Z 1432.858,A 0.000,B 0.000,C 90.000,E1 10.423} C_DIS
LIN {X -0.063,Y -366.744,Z 1432.858,A 0.000,B 0.000,C 90.000,E1 10.423} C_DIS
LIN {X -0.115,Y -366.496,Z 1432.855,A 0.000,B 0.000,C 90.000,E1 9.962} C_DIS
LIN {X 0.182,Y -361.797,Z 1432.822,A 0.000,B 0.000,C 90.000,E1 3.955} C_DIS
LIN {X 0.067,Y -360.903,Z 1432.801,A 0.000,B 0.000,C 90.000,E1 0.229} C_DIS
LIN {X -0.053,Y -359.426,Z 1432.770,A 0.000,B 0.000,C 90.000,E1 354.546} C_DIS
LIN {X 0.070,Y -358.890,Z 1432.759,A 0.000,B 0.000,C 90.000,E1 352.648} C_DIS
LIN {X -0.020,Y -359.563,Z 1432.726,A 0.000,B 0.000,C 90.000,E1 346.645} C_DIS
LIN {X 0.001,Y -361.801,Z 1432.684,A 0.000,B 0.000,C 90.000,E1 339.135} C_DIS
LIN {X -0.154,Y -362.053,Z 1432.680,A 0.000,B 0.000,C 90.000,E1 338.411} C_DIS
LIN {X 0.189,Y -365.980,Z 1432.643,A 0.000,B 0.000,C 90.000,E1 331.641} C_DIS
LIN {X 0.029,Y -366.387,Z 1432.639,A 0.000,B 0.000,C 90.000,E1 330.923} C_DIS
LIN {X -0.031,Y -371.355,Z 1432.604,A 0.000,B 0.000,C 90.000,E1 324.642} C_DIS
LIN {X -0.043,Y -371.766,Z 1432.602,A 0.000,B 0.000,C 90.000,E1 324.276} C_DIS
LIN {X 0.013,Y -377.358,Z 1432.567,A 0.000,B 0.000,C 90.000,E1 318.038} C_DIS
LIN {X 0.012,Y -378.235,Z 1432.563,A 0.000,B 0.000,C 90.000,E1 317.310} C_DIS
LIN {X 0.002,Y -383.940,Z 1432.531,A 0.000,B 0.000,C 90.000,E1 311.515} C_DIS
LIN {X 0.088,Y -384.893,Z 1432.527,A 0.000,B 0.000,C 90.000,E1 310.782} C_DIS
LIN {X 0.262,Y -390.610,Z 1432.495,A 0.000,B 0.000,C 90.000,E1 305.025} C_DIS
LIN {X 0.106,Y -391.104,Z 1432.493,A 0.000,B 0.000,C 90.000,E1 304.692} C_DIS
LIN {X 0.022,Y -391.648,Z 1432.489,A 0.000,B 0.000,C 90.000,E1 303.992} C_DIS
LIN {X -0.080,Y -396.825,Z 1432.459,A 0.000,B 0.000,C 90.000,E1 298.693} C_DIS
LIN {X -0.210,Y -397.120,Z 1432.457,A 0.000,B 0.000,C 90.000,E1 298.359} C_DIS
LIN {X -0.055,Y -401.597,Z 1432.426,A 0.000,B 0.000,C 90.000,E1 292.717} C_DIS
LIN {X 0.222,Y -404.659,Z 1432.395,A 0.000,B 0.000,C 90.000,E1 287.094} C_DIS
LIN {X -0.079,Y -404.735,Z 1432.391,A 0.000,B 0.000,C 90.000,E1 286.441} C_DIS
LIN {X 0.214,Y -406.099,Z 1432.364,A 0.000,B 0.000,C 90.000,E1 281.535} C_DIS
LIN {X -0.176,Y -406.094,Z 1432.362,A 0.000,B 0.000,C 90.000,E1 281.243} C_DIS
LIN {X -0.097,Y -405.680,Z 1432.333,A 0.000,B 0.000,C 90.000,E1 276.024} C_DIS
LIN {X -0.165,Y -405.058,Z 1432.328,A 0.000,B 0.000,C 90.000,E1 274.992} C_DIS
LIN {X -0.060,Y -403.497,Z 1432.304,A 0.000,B 0.000,C 90.000,E1 270.802} C_DIS
LIN {X -0.092,Y -403.288,Z 1432.302,A 0.000,B 0.000,C 90.000,E1 270.458} C_DIS
LIN {X 0.091,Y -398.931,Z 1432.271,A 0.000,B 0.000,C 90.000,E1 264.837} C_DIS
LIN {X -0.040,Y -393.108,Z 1432.242,A 0.000,B 0.000,C 90.000,E1 259.567} C_DIS
LIN {X -0.079,Y -392.835,Z 1432.240,A 0.000,B 0.000,C 90.000,E1 259.218} C_DIS
LIN {X 0.034,Y -385.993,Z 1432.212,A 0.000,B 0.000,C 90.000,E1 254.212} C_DIS
LIN {X -0.026,Y -385.267,Z 1432.208,A 0.000,B 0.000,C 90.000,E1 253.504} C_DIS
LIN {X -0.004,Y -384.768,Z 1432.206,A 0.000,B 0.000,C 90.000,E1 253.142} C_DIS
LIN {X 0.221,Y -377.973,Z 1432.182,A 0.000,B 0.000,C 90.000,E1 248.773} C_DIS
LIN {X -0.044,Y -376.233,Z 1432.174,A 0.000,B 0.000,C 90.000,E1 247.358} C_DIS
LIN {X 0.057,Y -374.944,Z 1432.170,A 0.000,B 0.000,C 90.000,E1 246.613} C_DIS
LIN {X -0.208,Y -368.417,Z 1432.148,A 0.000,B 0.000,C 90.000,E1 242.615} C_DIS
LIN {X 0.097,Y -366.047,Z 1432.137,A 0.000,B 0.000,C 90.000,E1 240.717} C_DIS
LIN {X 0.004,Y -359.196,Z 1432.115,A 0.000,B 0.000,C 90.000,E1 236.628} C_DIS
LIN {X 0.021,Y -355.842,Z 1432.100,A 0.000,B 0.000,C 90.000,E1 233.989} C_DIS
LIN {X -0.173,Y -348.793,Z 1432.075,A 0.000,B 0.000,C 90.000,E1 229.461} C_DIS
LIN {X -0.097,Y -346.185,Z 1432.062,A 0.000,B 0.000,C 90.000,E1 227.148} C_DIS
LIN {X -0.088,Y -345.065,Z 1432.058,A 0.000,B 0.000,C 90.000,E1 226.377} C_DIS
LIN {X 0.094,Y -338.586,Z 1432.030,A 0.000,B 0.000,C 90.000,E1 221.310} C_DIS
LIN {X 0.094,Y -336.840,Z 1432.019,A 0.000,B 0.000,C 90.000,E1 219.358} C_DIS
LIN {X 0.014,Y -330.861,Z 1431.988,A 0.000,B 0.000,C 90.000,E1 213.865} C_DIS
LIN {X 0.149,Y -329.296,Z 1431.975,A 0.000,B 0.000,C 90.000,E1 211.465} C_DIS
LIN {X -0.154,Y -324.669,Z 1431.942,A 0.000,B 0.000,C 90.000,E1 205.540} C_DIS
LIN {X 0.174,Y -323.837,Z 1431.928,A 0.000,B 0.000,C 90.000,E1 203.078} C_DIS
LIN {X -0.017,Y -321.124,Z 1431.881,A 0.000,B 0.000,C 90.000,E1 194.662} C_DIS
LIN {X 0.138,Y -320.932,Z 1431.877,A 0.000,B 0.000,C 90.000,E1 193.828} C_DIS
LIN {X -0.076,Y -321.562,Z 1431.832,A 0.000,B 0.000,C 90.000,E1 185.796} C_DIS
LIN {X -0.143,Y -324.415,Z 1431.790,A 0.000,B 0.000,C 90.000,E1 178.165} C_DIS
LIN {X -0.141,Y -325.376,Z 1431.783,A 0.000,B 0.000,C 90.000,E1 176.963} C_DIS
LIN {X -0.100,Y -329.112,Z 1431.750,A 0.000,B 0.000,C 90.000,E1 170.971} C_DIS
LIN {X -0.028,Y -332.020,Z 1431.735,A 0.000,B 0.000,C 90.000,E1 168.285} C_DIS
LIN {X -0.061,Y -349.445,Z 1431.735,A 0.000,B 0.000,C 90.000,E1 168.285} C_DIS
LIN {X 0.097,Y -350.841,Z 1431.735,A 0.000,B 0.000,C 90.000,E1 168.229} C_DIS
LIN {X 0.029,Y -352.515,Z 1431.734,A 0.000,B 0.000,C 90.000,E1 168.173} C_DIS
LIN {X -0.092,Y -355.061,Z 1431.734,A 0.000,B 0.000,C 90.000,E1 168.049} C_DIS
LIN {X 0.081,Y -357.866,Z 1431.733,A 0.000,B 0.000,C 90.000,E1 167.825} C_DIS
LIN {X 0.032,Y -362.380,Z 1431.730,A 0.000,B 0.000,C 90.000,E1 167.465} C_DIS
LIN {X 0.130,Y -368.413,Z 1431.727,A 0.000,B 0.000,C 90.000,E1 166.881} C_DIS
LIN {X -0.036,Y -374.394,Z 1431.724,A 0.000,B 0.000,C 90.000,E1 166.284} C_DIS
LIN {X -0.096,Y -389.266,Z 1431.715,A 0.000,B 0.000,C 90.000,E1 164.685} C_DIS
LIN {X -0.216,Y -399.706,Z 1431.709,A 0.000,B 0.000,C 90.000,E1 163.685} C_DIS
LIN {X 0.081,Y -416.706,Z 1431.701,A 0.000,B 0.000,C 90.000,E1 162.127} C_DIS
LIN {X 0.188,Y -430.731,Z 1431.694,A 0.000,B 0.000,C 90.000,E1 160.913} C_DIS
LIN {X 0.073,Y -444.714,Z 1431.688,A 0.000,B 0.000,C 90.000,E1 159.752} C_DIS
LIN {X 0.025,Y -460.060,Z 1431.680,A 0.000,B 0.000,C 90.000,E1 158.465} C_DIS
LIN {X -0.134,Y -469.127,Z 1431.676,A 0.000,B 0.000,C 90.000,E1 157.720} C_DIS
LIN {X 0.047,Y -480.954,Z 1431.670,A 0.000,B 0.000,C 90.000,E1 156.666} C_DIS
LIN {X -0.257,Y -486.678,Z 1431.667,A 0.000,B 0.000,C 90.000,E1 156.177} C_DIS
LIN {X -0.202,Y -496.626,Z 1431.662,A 0.000,B 0.000,C 90.000,E1 155.229} C_DIS
LIN {X -0.303,Y -504.728,Z 1431.658,A 0.000,B 0.000,C 90.000,E1 154.409} C_DIS
LIN {X 0.180,Y -511.312,Z 1431.654,A 0.000,B 0.000,C 90.000,E1 153.640} C_DIS
LIN {X 0.030,Y -517.184,Z 1431.650,A 0.000,B 0.000,C 90.000,E1 152.922} C_DIS
LIN {X -0.016,Y -520.523,Z 1431.647,A 0.000,B 0.000,C 90.000,E1 152.487} C_DIS
LIN {X 0.035,Y -524.540,Z 1431.644,A 0.000,B 0.000,C 90.000,E1 151.897} C_DIS
LIN {X 0.119,Y -528.047,Z 1431.641,A 0.000,B 0.000,C 90.000,E1 151.307} C_DIS
LIN {X 0.079,Y -532.000,Z 1431.637,A 0.000,B 0.000,C 90.000,E1 150.589} C_DIS
LIN {X 0.219,Y -534.749,Z 1431.634,A 0.000,B 0.000,C 90.000,E1 149.999} C_DIS
LIN {X -0.085,Y -537.263,Z 1431.630,A 0.000,B 0.000,C 90.000,E1 149.459} C_DIS
LIN {X 0.089,Y -539.494,Z 1431.627,A 0.000,B 0.000,C 90.000,E1 148.869} C_DIS
LIN {X 0.285,Y -542.365,Z 1431.622,A 0.000,B 0.000,C 90.000,E1 147.995} C_DIS
LIN {X 0.032,Y -544.099,Z 1431.619,A 0.000,B 0.000,C 90.000,E1 147.454} C_DIS
LIN {X -0.181,Y -546.438,Z 1431.615,A 0.000,B 0.000,C 90.000,E1 146.628} C_DIS
LIN {X 0.085,Y -548.469,Z 1431.610,A 0.000,B 0.000,C 90.000,E1 145.754} C_DIS
LIN {X 0.231,Y -550.325,Z 1431.605,A 0.000,B 0.000,C 90.000,E1 144.895} C_DIS
LIN {X 0.080,Y -551.973,Z 1431.600,A 0.000,B 0.000,C 90.000,E1 144.069} C_DIS
LIN {X -0.175,Y -553.258,Z 1431.596,A 0.000,B 0.000,C 90.000,E1 143.256} C_DIS
LIN {X 0.103,Y -554.715,Z 1431.590,A 0.000,B 0.000,C 90.000,E1 142.110} C_DIS
LIN {X -0.036,Y -555.952,Z 1431.583,A 0.000,B 0.000,C 90.000,E1 141.009} C_DIS
LIN {X -0.162,Y -556.945,Z 1431.577,A 0.000,B 0.000,C 90.000,E1 139.908} C_DIS
LIN {X 0.160,Y -558.023,Z 1431.569,A 0.000,B 0.000,C 90.000,E1 138.485} C_DIS
LIN {X 0.002,Y -558.778,Z 1431.563,A 0.000,B 0.000,C 90.000,E1 137.391} C_DIS
LIN {X -0.143,Y -559.510,Z 1431.557,A 0.000,B 0.000,C 90.000,E1 136.296} C_DIS
LIN {X 0.110,Y -560.027,Z 1431.551,A 0.000,B 0.000,C 90.000,E1 135.162} C_DIS
LIN {X 0.372,Y -560.420,Z 1431.545,A 0.000,B 0.000,C 90.000,E1 134.028} C_DIS
LIN {X 0.251,Y -560.752,Z 1431.539,A 0.000,B 0.000,C 90.000,E1 132.933} C_DIS
LIN {X 0.134,Y -560.964,Z 1431.533,A 0.000,B 0.000,C 90.000,E1 131.838} C_DIS
LIN {X -0.143,Y -561.054,Z 1431.522,A 0.000,B 0.000,C 90.000,E1 129.930} C_DIS
LIN {X -0.105,Y -561.139,Z 1431.514,A 0.000,B 0.000,C 90.000,E1 128.543} C_DIS
LIN {X 0.035,Y -561.116,Z 1431.505,A 0.000,B 0.000,C 90.000,E1 126.870} C_DIS
LIN {X -0.075,Y -560.961,Z 1431.494,A 0.000,B 0.000,C 90.000,E1 124.945} C_DIS
LIN {X -0.239,Y -560.744,Z 1431.486,A 0.000,B 0.000,C 90.000,E1 123.579} C_DIS
LIN {X 0.073,Y -560.485,Z 1431.479,A 0.000,B 0.000,C 90.000,E1 122.163} C_DIS
LIN {X 0.075,Y -560.666,Z 1431.459,A 0.000,B 0.000,C 90.000,E1 118.565} C_DIS
LIN {X -0.008,Y -561.388,Z 1431.447,A 0.000,B 0.000,C 90.000,E1 116.360} C_DIS
LIN {X 0.018,Y -561.934,Z 1431.439,A 0.000,B 0.000,C 90.000,E1 114.975} C_DIS
LIN {X 0.060,Y -562.270,Z 1431.431,A 0.000,B 0.000,C 90.000,E1 113.590} C_DIS
LIN {X -0.105,Y -563.020,Z 1431.422,A 0.000,B 0.000,C 90.000,E1 111.950} C_DIS
LIN {X 0.228,Y -564.030,Z 1431.418,A 0.000,B 0.000,C 90.000,E1 111.227} C_DIS
LIN {X -0.076,Y -565.326,Z 1431.416,A 0.000,B 0.000,C 90.000,E1 110.844} C_DIS
LIN {X 0.132,Y -568.044,Z 1431.414,A 0.000,B 0.000,C 90.000,E1 110.556} C_DIS
LIN {X 0.213,Y -568.596,Z 1431.414,A 0.000,B 0.000,C 90.000,E1 110.482} C_DIS
LIN {X -0.087,Y -578.109,Z 1431.411,A 0.000,B 0.000,C 90.000,E1 109.939} C_DIS
LIN {X -0.327,Y -584.028,Z 1431.409,A 0.000,B 0.000,C 90.000,E1 109.577} C_DIS
LIN {X -0.138,Y -589.685,Z 1431.406,A 0.000,B 0.000,C 90.000,E1 109.141} C_DIS
LIN {X 0.073,Y -594.746,Z 1431.404,A 0.000,B 0.000,C 90.000,E1 108.671} C_DIS
LIN {X 0.053,Y -600.874,Z 1431.400,A 0.000,B 0.000,C 90.000,E1 108.055} C_DIS
LIN {X -0.366,Y -605.101,Z 1431.398,A 0.000,B 0.000,C 90.000,E1 107.583} C_DIS
LIN {X -0.151,Y -609.040,Z 1431.395,A 0.000,B 0.000,C 90.000,E1 107.040} C_DIS
LIN {X -0.121,Y -613.053,Z 1431.391,A 0.000,B 0.000,C 90.000,E1 106.386} C_DIS
LIN {X -0.198,Y -614.279,Z 1431.390,A 0.000,B 0.000,C 90.000,E1 106.134} C_DIS
LIN {X -0.091,Y -616.334,Z 1431.387,A 0.000,B 0.000,C 90.000,E1 105.607} C_DIS
LIN {X 0.195,Y -617.742,Z 1431.384,A 0.000,B 0.000,C 90.000,E1 105.064} C_DIS
LIN {X 0.104,Y -619.090,Z 1431.380,A 0.000,B 0.000,C 90.000,E1 104.300} C_DIS
LIN {X 0.031,Y -620.303,Z 1431.375,A 0.000,B 0.000,C 90.000,E1 103.536} C_DIS
LIN {X 0.192,Y -620.902,Z 1431.372,A 0.000,B 0.000,C 90.000,E1 103.008} C_DIS
LIN {X 0.140,Y -621.296,Z 1431.368,A 0.000,B 0.000,C 90.000,E1 102.243} C_DIS
LIN {X -0.081,Y -621.382,Z 1431.367,A 0.000,B 0.000,C 90.000,E1 102.007} C_DIS
LIN {X -0.133,Y -621.060,Z 1431.362,A 0.000,B 0.000,C 90.000,E1 101.243} C_DIS
LIN {X 0.030,Y -620.519,Z 1431.360,A 0.000,B 0.000,C 90.000,E1 100.715} C_DIS
LIN {X 0.077,Y -619.513,Z 1431.357,A 0.000,B 0.000,C 90.000,E1 100.197} C_DIS
LIN {X -0.107,Y -617.615,Z 1431.352,A 0.000,B 0.000,C 90.000,E1 99.443} C_DIS
LIN {X 0.029,Y -616.018,Z 1431.350,A 0.000,B 0.000,C 90.000,E1 98.916} C_DIS
LIN {X 0.057,Y -614.063,Z 1431.347,A 0.000,B 0.000,C 90.000,E1 98.398} C_DIS
LIN {X -0.011,Y -611.158,Z 1431.343,A 0.000,B 0.000,C 90.000,E1 97.757} C_DIS
LIN {X 0.316,Y -607.091,Z 1431.339,A 0.000,B 0.000,C 90.000,E1 96.947} C_DIS
LIN {X -0.075,Y -602.516,Z 1431.334,A 0.000,B 0.000,C 90.000,E1 96.201} C_DIS
LIN {X -0.135,Y -599.151,Z 1431.332,A 0.000,B 0.000,C 90.000,E1 95.682} C_DIS
LIN {X 0.151,Y -597.014,Z 1431.330,A 0.000,B 0.000,C 90.000,E1 95.391} C_DIS
LIN {X 0.187,Y -593.517,Z 1431.328,A 0.000,B 0.000,C 90.000,E1 94.992} C_DIS
LIN {X -0.141,Y -590.780,Z 1431.326,A 0.000,B 0.000,C 90.000,E1 94.759} C_DIS
LIN {X 0.181,Y -585.130,Z 1431.324,A 0.000,B 0.000,C 90.000,E1 94.245} C_DIS
LIN {X -0.131,Y -577.872,Z 1431.321,A 0.000,B 0.000,C 90.000,E1 93.726} C_DIS
LIN {X -0.242,Y -573.956,Z 1431.319,A 0.000,B 0.000,C 90.000,E1 93.383} C_DIS
LIN {X 0.201,Y -572.524,Z 1431.318,A 0.000,B 0.000,C 90.000,E1 93.154} C_DIS
LIN {X 0.164,Y -572.089,Z 1431.317,A 0.000,B 0.000,C 90.000,E1 93.037} C_DIS
LIN {X -0.055,Y -571.802,Z 1431.316,A 0.000,B 0.000,C 90.000,E1 92.922} C_DIS
LIN {X -0.139,Y -571.416,Z 1431.314,A 0.000,B 0.000,C 90.000,E1 92.522} C_DIS
LIN {X 0.130,Y -571.472,Z 1431.311,A 0.000,B 0.000,C 90.000,E1 91.949} C_DIS
LIN {X -0.190,Y -573.718,Z 1431.296,A 0.000,B 0.000,C 90.000,E1 89.255} C_DIS
LIN {X -0.026,Y -574.965,Z 1431.288,A 0.000,B 0.000,C 90.000,E1 87.879} C_DIS
LIN {X -0.263,Y -576.498,Z 1431.279,A 0.000,B 0.000,C 90.000,E1 86.274} C_DIS
LIN {X 0.132,Y -578.056,Z 1431.270,A 0.000,B 0.000,C 90.000,E1 84.609} C_DIS
LIN {X 0.035,Y -579.684,Z 1431.261,A 0.000,B 0.000,C 90.000,E1 82.996} C_DIS
LIN {X 0.043,Y -581.405,Z 1431.252,A 0.000,B 0.000,C 90.000,E1 81.376} C_DIS
LIN {X -0.153,Y -583.370,Z 1431.242,A 0.000,B 0.000,C 90.000,E1 79.511} C_DIS
LIN {X 0.029,Y -585.071,Z 1431.233,A 0.000,B 0.000,C 90.000,E1 77.881} C_DIS
LIN {X -0.137,Y -585.950,Z 1431.227,A 0.000,B 0.000,C 90.000,E1 76.825} C_DIS
LIN {X 0.095,Y -587.007,Z 1431.219,A 0.000,B 0.000,C 90.000,E1 75.463} C_DIS
LIN {X 0.026,Y -588.058,Z 1431.210,A 0.000,B 0.000,C 90.000,E1 73.866} C_DIS
LIN {X -0.109,Y -588.796,Z 1431.203,A 0.000,B 0.000,C 90.000,E1 72.543} C_DIS
LIN {X 0.198,Y -589.604,Z 1431.194,A 0.000,B 0.000,C 90.000,E1 70.913} C_DIS
LIN {X -0.041,Y -590.531,Z 1431.185,A 0.000,B 0.000,C 90.000,E1 69.337} C_DIS
LIN {X 0.163,Y -591.409,Z 1431.176,A 0.000,B 0.000,C 90.000,E1 67.720} C_DIS
LIN {X 0.157,Y -592.445,Z 1431.167,A 0.000,B 0.000,C 90.000,E1 66.125} C_DIS
LIN {X -0.090,Y -593.847,Z 1431.156,A 0.000,B 0.000,C 90.000,E1 64.024} C_DIS
LIN {X -0.022,Y -594.932,Z 1431.148,A 0.000,B 0.000,C 90.000,E1 62.692} C_DIS
LIN {X -0.084,Y -596.359,Z 1431.138,A 0.000,B 0.000,C 90.000,E1 60.845} C_DIS
LIN {X -0.226,Y -597.549,Z 1431.131,A 0.000,B 0.000,C 90.000,E1 59.537} C_DIS
LIN {X 0.088,Y -599.253,Z 1431.120,A 0.000,B 0.000,C 90.000,E1 57.661} C_DIS
LIN {X 0.260,Y -600.922,Z 1431.110,A 0.000,B 0.000,C 90.000,E1 55.801} C_DIS
LIN {X -0.275,Y -602.301,Z 1431.101,A 0.000,B 0.000,C 90.000,E1 54.276} C_DIS
LIN {X 0.149,Y -603.354,Z 1431.094,A 0.000,B 0.000,C 90.000,E1 52.924} C_DIS
LIN {X -0.104,Y -604.454,Z 1431.085,A 0.000,B 0.000,C 90.000,E1 51.376} C_DIS
LIN {X 0.132,Y -605.380,Z 1431.077,A 0.000,B 0.000,C 90.000,E1 49.784} C_DIS
LIN {X 0.042,Y -605.672,Z 1431.069,A 0.000,B 0.000,C 90.000,E1 48.485} C_DIS
LIN {X -0.020,Y -605.920,Z 1431.059,A 0.000,B 0.000,C 90.000,E1 46.662} C_DIS
LIN {X 0.124,Y -605.987,Z 1431.051,A 0.000,B 0.000,C 90.000,E1 45.081} C_DIS
LIN {X 0.021,Y -605.585,Z 1431.043,A 0.000,B 0.000,C 90.000,E1 43.785} C_DIS
LIN {X 0.074,Y -605.368,Z 1431.040,A 0.000,B 0.000,C 90.000,E1 43.257} C_DIS
LIN {X -0.054,Y -604.529,Z 1431.033,A 0.000,B 0.000,C 90.000,E1 41.962} C_DIS
LIN {X 0.041,Y -603.679,Z 1431.027,A 0.000,B 0.000,C 90.000,E1 40.906} C_DIS
LIN {X 0.377,Y -602.318,Z 1431.020,A 0.000,B 0.000,C 90.000,E1 39.564} C_DIS
LIN {X -0.185,Y -601.389,Z 1431.016,A 0.000,B 0.000,C 90.000,E1 38.830} C_DIS
LIN {X -0.263,Y -599.553,Z 1431.008,A 0.000,B 0.000,C 90.000,E1 37.523} C_DIS
LIN {X 0.225,Y -598.758,Z 1431.005,A 0.000,B 0.000,C 90.000,E1 36.950} C_DIS
LIN {X 0.091,Y -596.284,Z 1430.998,A 0.000,B 0.000,C 90.000,E1 35.644} C_DIS
LIN {X -0.058,Y -594.610,Z 1430.994,A 0.000,B 0.000,C 90.000,E1 34.865} C_DIS
LIN {X -0.069,Y -592.775,Z 1430.989,A 0.000,B 0.000,C 90.000,E1 34.072} C_DIS
LIN {X -0.050,Y -590.076,Z 1430.983,A 0.000,B 0.000,C 90.000,E1 33.007} C_DIS
LIN {X -0.092,Y -587.834,Z 1430.979,A 0.000,B 0.000,C 90.000,E1 32.212} C_DIS
LIN {X 0.097,Y -587.047,Z 1430.977,A 0.000,B 0.000,C 90.000,E1 31.926} C_DIS
LIN {X -0.101,Y -583.265,Z 1430.972,A 0.000,B 0.000,C 90.000,E1 30.875} C_DIS
LIN {X 0.088,Y -580.019,Z 1430.967,A 0.000,B 0.000,C 90.000,E1 30.050} C_DIS
LIN {X -0.054,Y -576.443,Z 1430.963,A 0.000,B 0.000,C 90.000,E1 29.255} C_DIS
LIN {X 0.149,Y -573.849,Z 1430.960,A 0.000,B 0.000,C 90.000,E1 28.693} C_DIS
LIN {X -0.088,Y -571.764,Z 1430.957,A 0.000,B 0.000,C 90.000,E1 28.309} C_DIS
LIN {X -0.234,Y -567.993,Z 1430.953,A 0.000,B 0.000,C 90.000,E1 27.641} C_DIS
LIN {X -0.106,Y -562.435,Z 1430.948,A 0.000,B 0.000,C 90.000,E1 26.668} C_DIS
LIN {X 0.203,Y -556.290,Z 1430.943,A 0.000,B 0.000,C 90.000,E1 25.668} C_DIS
LIN {X 0.055,Y -550.620,Z 1430.938,A 0.000,B 0.000,C 90.000,E1 24.847} C_DIS
LIN {X -0.292,Y -547.646,Z 1430.936,A 0.000,B 0.000,C 90.000,E1 24.463} C_DIS
LIN {X -0.276,Y -543.386,Z 1430.933,A 0.000,B 0.000,C 90.000,E1 23.898} C_DIS
LIN {X 0.072,Y -537.600,Z 1430.929,A 0.000,B 0.000,C 90.000,E1 23.153} C_DIS
LIN {X -0.032,Y -531.582,Z 1430.925,A 0.000,B 0.000,C 90.000,E1 22.461} C_DIS
LIN {X -0.128,Y -526.525,Z 1430.922,A 0.000,B 0.000,C 90.000,E1 21.897} C_DIS
LIN {X -0.238,Y -516.136,Z 1430.915,A 0.000,B 0.000,C 90.000,E1 20.791} C_DIS
LIN {X -0.229,Y -506.790,Z 1430.910,A 0.000,B 0.000,C 90.000,E1 19.812} C_DIS
LIN {X 0.184,Y -496.195,Z 1430.904,A 0.000,B 0.000,C 90.000,E1 18.671} C_DIS
LIN {X 0.115,Y -478.620,Z 1430.894,A 0.000,B 0.000,C 90.000,E1 16.858} C_DIS
LIN {X -0.103,Y -466.422,Z 1430.886,A 0.000,B 0.000,C 90.000,E1 15.552} C_DIS
LIN {X 0.210,Y -451.604,Z 1430.877,A 0.000,B 0.000,C 90.000,E1 13.828} C_DIS
LIN {X 0.102,Y -435.564,Z 1430.867,A 0.000,B 0.000,C 90.000,E1 11.951} C_DIS
LIN {X -0.003,Y -431.296,Z 1430.864,A 0.000,B 0.000,C 90.000,E1 11.478} C_DIS
LIN {X 0.168,Y -425.285,Z 1430.860,A 0.000,B 0.000,C 90.000,E1 10.838} C_DIS
LIN {X -0.072,Y -420.611,Z 1430.858,A 0.000,B 0.000,C 90.000,E1 10.433} C_DIS
LIN {X 0.045,Y -417.288,Z 1430.856,A 0.000,B 0.000,C 90.000,E1 10.141} C_DIS
LIN {X -0.088,Y -413.673,Z 1430.855,A 0.000,B 0.000,C 90.000,E1 9.905} C_DIS
LIN {X 0.056,Y -410.735,Z 1430.854,A 0.000,B 0.000,C 90.000,E1 9.726} C_DIS
LIN {X -0.116,Y -408.111,Z 1430.854,A 0.000,B 0.000,C 90.000,E1 9.670} C_DIS
LIN {X -0.143,Y -407.716,Z 1430.854,A 0.000,B 0.000,C 90.000,E1 9.670} C_DIS
LIN {X -0.152,Y -366.212,Z 1430.854,A 0.000,B 0.000,C 90.000,E1 9.670} C_DIS
LIN {X 0.023,Y -361.639,Z 1430.820,A 0.000,B 0.000,C 90.000,E1 3.612} C_DIS
LIN {X 0.105,Y -360.903,Z 1430.801,A 0.000,B 0.000,C 90.000,E1 0.229} C_DIS
LIN {X -0.053,Y -359.426,Z 1430.770,A 0.000,B 0.000,C 90.000,E1 354.546} C_DIS
LIN {X 0.070,Y -358.890,Z 1430.759,A 0.000,B 0.000,C 90.000,E1 352.648} C_DIS
LIN {X -0.020,Y -359.563,Z 1430.726,A 0.000,B 0.000,C 90.000,E1 346.645} C_DIS
LIN {X 0.001,Y -361.801,Z 1430.684,A 0.000,B 0.000,C 90.000,E1 339.135} C_DIS
LIN {X -0.154,Y -362.053,Z 1430.680,A 0.000,B 0.000,C 90.000,E1 338.411} C_DIS
LIN {X 0.189,Y -365.980,Z 1430.643,A 0.000,B 0.000,C 90.000,E1 331.641} C_DIS
LIN {X 0.029,Y -366.387,Z 1430.639,A 0.000,B 0.000,C 90.000,E1 330.923} C_DIS
LIN {X -0.031,Y -371.355,Z 1430.604,A 0.000,B 0.000,C 90.000,E1 324.642} C_DIS
LIN {X -0.043,Y -371.766,Z 1430.602,A 0.000,B 0.000,C 90.000,E1 324.276} C_DIS
LIN {X 0.013,Y -377.358,Z 1430.567,A 0.000,B 0.000,C 90.000,E1 318.038} C_DIS
LIN {X 0.012,Y -378.235,Z 1430.563,A 0.000,B 0.000,C 90.000,E1 317.310} C_DIS
LIN {X 0.002,Y -383.940,Z 1430.531,A 0.000,B 0.000,C 90.000,E1 311.515} C_DIS
LIN {X 0.088,Y -384.893,Z 1430.527,A 0.000,B 0.000,C 90.000,E1 310.782} C_DIS
LIN {X 0.262,Y -390.610,Z 1430.495,A 0.000,B 0.000,C 90.000,E1 305.025} C_DIS
LIN {X 0.106,Y -391.104,Z 1430.493,A 0.000,B 0.000,C 90.000,E1 304.692} C_DIS
LIN {X 0.022,Y -391.648,Z 1430.489,A 0.000,B 0.000,C 90.000,E1 303.992} C_DIS
LIN {X -0.080,Y -396.825,Z 1430.459,A 0.000,B 0.000,C 90.000,E1 298.693} C_DIS
LIN {X -0.210,Y -397.120,Z 1430.457,A 0.000,B 0.000,C 90.000,E1 298.359} C_DIS
LIN {X -0.055,Y -401.597,Z 1430.426,A 0.000,B 0.000,C 90.000,E1 292.717} C_DIS
LIN {X 0.222,Y -404.659,Z 1430.395,A 0.000,B 0.000,C 90.000,E1 287.094} C_DIS
LIN {X -0.079,Y -404.735,Z 1430.391,A 0.000,B 0.000,C 90.000,E1 286.441} C_DIS
LIN {X 0.214,Y -406.099,Z 1430.364,A 0.000,B 0.000,C 90.000,E1 281.535} C_DIS
LIN {X -0.176,Y -406.094,Z 1430.362,A 0.000,B 0.000,C 90.000,E1 281.243} C_DIS
LIN {X -0.097,Y -405.680,Z 1430.333,A 0.000,B 0.000,C 90.000,E1 276.024} C_DIS
LIN {X -0.165,Y -405.058,Z 1430.328,A 0.000,B 0.000,C 90.000,E1 274.992} C_DIS
LIN {X -0.060,Y -403.497,Z 1430.304,A 0.000,B 0.000,C 90.000,E1 270.802} C_DIS
LIN {X -0.092,Y -403.288,Z 1430.302,A 0.000,B 0.000,C 90.000,E1 270.458} C_DIS
LIN {X 0.091,Y -398.931,Z 1430.271,A 0.000,B 0.000,C 90.000,E1 264.837} C_DIS
LIN {X -0.040,Y -393.108,Z 1430.242,A 0.000,B 0.000,C 90.000,E1 259.567} C_DIS
LIN {X -0.079,Y -392.835,Z 1430.240,A 0.000,B 0.000,C 90.000,E1 259.218} C_DIS
LIN {X 0.034,Y -385.993,Z 1430.212,A 0.000,B 0.000,C 90.000,E1 254.212} C_DIS
LIN {X -0.026,Y -385.267,Z 1430.208,A 0.000,B 0.000,C 90.000,E1 253.504} C_DIS
LIN {X -0.004,Y -384.768,Z 1430.206,A 0.000,B 0.000,C 90.000,E1 253.142} C_DIS
LIN {X 0.221,Y -377.973,Z 1430.182,A 0.000,B 0.000,C 90.000,E1 248.773} C_DIS
LIN {X -0.044,Y -376.233,Z 1430.174,A 0.000,B 0.000,C 90.000,E1 247.358} C_DIS
LIN {X 0.057,Y -374.944,Z 1430.170,A 0.000,B 0.000,C 90.000,E1 246.613} C_DIS
LIN {X -0.208,Y -368.417,Z 1430.148,A 0.000,B 0.000,C 90.000,E1 242.615} C_DIS
LIN {X 0.097,Y -366.047,Z 1430.137,A 0.000,B 0.000,C 90.000,E1 240.717} C_DIS
LIN {X 0.004,Y -359.196,Z 1430.115,A 0.000,B 0.000,C 90.000,E1 236.628} C_DIS
LIN {X 0.021,Y -355.842,Z 1430.100,A 0.000,B 0.000,C 90.000,E1 233.989} C_DIS
LIN {X -0.173,Y -348.793,Z 1430.075,A 0.000,B 0.000,C 90.000,E1 229.461} C_DIS
LIN {X -0.097,Y -346.185,Z 1430.062,A 0.000,B 0.000,C 90.000,E1 227.148} C_DIS
LIN {X -0.088,Y -345.065,Z 1430.058,A 0.000,B 0.000,C 90.000,E1 226.377} C_DIS
LIN {X 0.094,Y -338.586,Z 1430.030,A 0.000,B 0.000,C 90.000,E1 221.310} C_DIS
LIN {X 0.094,Y -336.840,Z 1430.019,A 0.000,B 0.000,C 90.000,E1 219.358} C_DIS
LIN {X 0.014,Y -330.861,Z 1429.988,A 0.000,B 0.000,C 90.000,E1 213.865} C_DIS
LIN {X 0.149,Y -329.296,Z 1429.975,A 0.000,B 0.000,C 90.000,E1 211.465} C_DIS
LIN {X -0.154,Y -324.669,Z 1429.942,A 0.000,B 0.000,C 90.000,E1 205.540} C_DIS
LIN {X 0.174,Y -323.837,Z 1429.928,A 0.000,B 0.000,C 90.000,E1 203.078} C_DIS
LIN {X -0.017,Y -321.124,Z 1429.881,A 0.000,B 0.000,C 90.000,E1 194.662} C_DIS
LIN {X 0.138,Y -320.932,Z 1429.877,A 0.000,B 0.000,C 90.000,E1 193.828} C_DIS
LIN {X -0.076,Y -321.562,Z 1429.832,A 0.000,B 0.000,C 90.000,E1 185.796} C_DIS
LIN {X -0.143,Y -324.415,Z 1429.790,A 0.000,B 0.000,C 90.000,E1 178.165} C_DIS
LIN {X -0.141,Y -325.376,Z 1429.783,A 0.000,B 0.000,C 90.000,E1 176.963} C_DIS
LIN {X -0.100,Y -329.112,Z 1429.750,A 0.000,B 0.000,C 90.000,E1 170.971} C_DIS
LIN {X -0.037,Y -330.981,Z 1429.740,A 0.000,B 0.000,C 90.000,E1 169.162} C_DIS
LIN {X -0.062,Y -343.190,Z 1429.740,A 0.000,B 0.000,C 90.000,E1 169.162} C_DIS
LIN {X 0.055,Y -346.096,Z 1429.739,A 0.000,B 0.000,C 90.000,E1 169.050} C_DIS
LIN {X -0.145,Y -347.751,Z 1429.739,A 0.000,B 0.000,C 90.000,E1 168.993} C_DIS
LIN {X 0.140,Y -350.566,Z 1429.738,A 0.000,B 0.000,C 90.000,E1 168.757} C_DIS
LIN {X 0.052,Y -354.931,Z 1429.736,A 0.000,B 0.000,C 90.000,E1 168.409} C_DIS
LIN {X 0.073,Y -360.972,Z 1429.732,A 0.000,B 0.000,C 90.000,E1 167.825} C_DIS
LIN {X 0.191,Y -366.956,Z 1429.729,A 0.000,B 0.000,C 90.000,E1 167.173} C_DIS
LIN {X -0.002,Y -372.801,Z 1429.725,A 0.000,B 0.000,C 90.000,E1 166.533} C_DIS
LIN {X -0.074,Y -381.645,Z 1429.719,A 0.000,B 0.000,C 90.000,E1 165.519} C_DIS
LIN {X 0.222,Y -393.836,Z 1429.713,A 0.000,B 0.000,C 90.000,E1 164.212} C_DIS
LIN {X -0.076,Y -412.551,Z 1429.703,A 0.000,B 0.000,C 90.000,E1 162.543} C_DIS
LIN {X 0.133,Y -429.772,Z 1429.695,A 0.000,B 0.000,C 90.000,E1 161.040} C_DIS
LIN {X 0.087,Y -445.194,Z 1429.688,A 0.000,B 0.000,C 90.000,E1 159.752} C_DIS
LIN {X 0.015,Y -459.011,Z 1429.681,A 0.000,B 0.000,C 90.000,E1 158.592} C_DIS
LIN {X -0.125,Y -469.576,Z 1429.676,A 0.000,B 0.000,C 90.000,E1 157.720} C_DIS
LIN {X 0.107,Y -481.309,Z 1429.671,A 0.000,B 0.000,C 90.000,E1 156.666} C_DIS
LIN {X -0.254,Y -487.105,Z 1429.667,A 0.000,B 0.000,C 90.000,E1 156.177} C_DIS
LIN {X -0.237,Y -497.070,Z 1429.662,A 0.000,B 0.000,C 90.000,E1 155.229} C_DIS
LIN {X 0.110,Y -505.145,Z 1429.658,A 0.000,B 0.000,C 90.000,E1 154.357} C_DIS
LIN {X 0.179,Y -511.664,Z 1429.654,A 0.000,B 0.000,C 90.000,E1 153.640} C_DIS
LIN {X 0.046,Y -517.514,Z 1429.650,A 0.000,B 0.000,C 90.000,E1 152.922} C_DIS
LIN {X 0.000,Y -520.833,Z 1429.647,A 0.000,B 0.000,C 90.000,E1 152.487} C_DIS
LIN {X 0.054,Y -524.850,Z 1429.644,A 0.000,B 0.000,C 90.000,E1 151.897} C_DIS
LIN {X -0.013,Y -529.154,Z 1429.640,A 0.000,B 0.000,C 90.000,E1 151.179} C_DIS
LIN {X 0.253,Y -531.590,Z 1429.638,A 0.000,B 0.000,C 90.000,E1 150.717} C_DIS
LIN {X 0.246,Y -535.037,Z 1429.634,A 0.000,B 0.000,C 90.000,E1 149.999} C_DIS
LIN {X -0.197,Y -538.102,Z 1429.630,A 0.000,B 0.000,C 90.000,E1 149.331} C_DIS
LIN {X -0.020,Y -540.281,Z 1429.626,A 0.000,B 0.000,C 90.000,E1 148.742} C_DIS
LIN {X -0.291,Y -542.187,Z 1429.623,A 0.000,B 0.000,C 90.000,E1 148.201} C_DIS
LIN {X -0.068,Y -544.725,Z 1429.619,A 0.000,B 0.000,C 90.000,E1 147.327} C_DIS
LIN {X -0.010,Y -546.314,Z 1429.615,A 0.000,B 0.000,C 90.000,E1 146.755} C_DIS
LIN {X 0.259,Y -548.373,Z 1429.611,A 0.000,B 0.000,C 90.000,E1 145.881} C_DIS
LIN {X 0.142,Y -550.794,Z 1429.604,A 0.000,B 0.000,C 90.000,E1 144.769} C_DIS
LIN {X 0.318,Y -552.379,Z 1429.600,A 0.000,B 0.000,C 90.000,E1 143.909} C_DIS
LIN {X -0.193,Y -553.935,Z 1429.594,A 0.000,B 0.000,C 90.000,E1 142.844} C_DIS
LIN {X 0.090,Y -555.313,Z 1429.587,A 0.000,B 0.000,C 90.000,E1 141.698} C_DIS
LIN {X 0.026,Y -556.680,Z 1429.580,A 0.000,B 0.000,C 90.000,E1 140.312} C_DIS
LIN {X -0.009,Y -557.973,Z 1429.570,A 0.000,B 0.000,C 90.000,E1 138.647} C_DIS
LIN {X -0.170,Y -558.721,Z 1429.564,A 0.000,B 0.000,C 90.000,E1 137.553} C_DIS
LIN {X 0.139,Y -559.570,Z 1429.556,A 0.000,B 0.000,C 90.000,E1 136.134} C_DIS
LIN {X -0.001,Y -560.078,Z 1429.550,A 0.000,B 0.000,C 90.000,E1 135.040} C_DIS
LIN {X -0.061,Y -560.558,Z 1429.543,A 0.000,B 0.000,C 90.000,E1 133.662} C_DIS
LIN {X -0.128,Y -560.870,Z 1429.535,A 0.000,B 0.000,C 90.000,E1 132.285} C_DIS
LIN {X 0.083,Y -560.931,Z 1429.530,A 0.000,B 0.000,C 90.000,E1 131.434} C_DIS
LIN {X 0.227,Y -561.062,Z 1429.520,A 0.000,B 0.000,C 90.000,E1 129.483} C_DIS
LIN {X 0.266,Y -561.100,Z 1429.512,A 0.000,B 0.000,C 90.000,E1 128.096} C_DIS
LIN {X -0.033,Y -561.090,Z 1429.504,A 0.000,B 0.000,C 90.000,E1 126.744} C_DIS
LIN {X -0.232,Y -560.973,Z 1429.495,A 0.000,B 0.000,C 90.000,E1 125.105} C_DIS
LIN {X -0.078,Y -560.789,Z 1429.487,A 0.000,B 0.000,C 90.000,E1 123.706} C_DIS
LIN {X -0.243,Y -560.523,Z 1429.480,A 0.000,B 0.000,C 90.000,E1 122.339} C_DIS
LIN {X -0.060,Y -560.569,Z 1429.461,A 0.000,B 0.000,C 90.000,E1 118.999} C_DIS
LIN {X 0.144,Y -561.359,Z 1429.447,A 0.000,B 0.000,C 90.000,E1 116.488} C_DIS
LIN {X -0.340,Y -561.924,Z 1429.440,A 0.000,B 0.000,C 90.000,E1 115.155} C_DIS
LIN {X -0.106,Y -562.182,Z 1429.433,A 0.000,B 0.000,C 90.000,E1 114.027} C_DIS
LIN {X 0.251,Y -562.864,Z 1429.424,A 0.000,B 0.000,C 90.000,E1 112.333} C_DIS
LIN {X 0.050,Y -563.068,Z 1429.423,A 0.000,B 0.000,C 90.000,E1 112.078} C_DIS
LIN {X 0.145,Y -563.928,Z 1429.419,A 0.000,B 0.000,C 90.000,E1 111.482} C_DIS
LIN {X -0.243,Y -565.256,Z 1429.418,A 0.000,B 0.000,C 90.000,E1 111.280} C_DIS
LIN {X 0.203,Y -565.937,Z 1429.417,A 0.000,B 0.000,C 90.000,E1 111.046} C_DIS
LIN {X -0.105,Y -568.326,Z 1429.416,A 0.000,B 0.000,C 90.000,E1 110.865} C_DIS
LIN {X -0.092,Y -570.076,Z 1429.415,A 0.000,B 0.000,C 90.000,E1 110.737} C_DIS
LIN {X -0.161,Y -579.014,Z 1429.412,A 0.000,B 0.000,C 90.000,E1 110.248} C_DIS
LIN {X -0.136,Y -584.623,Z 1429.410,A 0.000,B 0.000,C 90.000,E1 109.885} C_DIS
LIN {X 0.047,Y -590.126,Z 1429.408,A 0.000,B 0.000,C 90.000,E1 109.450} C_DIS
LIN {X 0.368,Y -595.454,Z 1429.406,A 0.000,B 0.000,C 90.000,E1 108.960} C_DIS
LIN {X -0.190,Y -599.200,Z 1429.404,A 0.000,B 0.000,C 90.000,E1 108.652} C_DIS
LIN {X -0.033,Y -603.954,Z 1429.401,A 0.000,B 0.000,C 90.000,E1 108.127} C_DIS
LIN {X -0.128,Y -606.287,Z 1429.399,A 0.000,B 0.000,C 90.000,E1 107.873} C_DIS
LIN {X -0.127,Y -611.171,Z 1429.396,A 0.000,B 0.000,C 90.000,E1 107.221} C_DIS
LIN {X 0.133,Y -614.446,Z 1429.393,A 0.000,B 0.000,C 90.000,E1 106.677} C_DIS
LIN {X -0.144,Y -616.561,Z 1429.391,A 0.000,B 0.000,C 90.000,E1 106.315} C_DIS
LIN {X -0.054,Y -619.183,Z 1429.387,A 0.000,B 0.000,C 90.000,E1 105.662} C_DIS
LIN {X -0.283,Y -619.864,Z 1429.386,A 0.000,B 0.000,C 90.000,E1 105.426} C_DIS
LIN {X -0.133,Y -620.965,Z 1429.383,A 0.000,B 0.000,C 90.000,E1 104.898} C_DIS
LIN {X -0.034,Y -622.225,Z 1429.378,A 0.000,B 0.000,C 90.000,E1 104.120} C_DIS
LIN {X -0.291,Y -623.625,Z 1429.373,A 0.000,B 0.000,C 90.000,E1 103.119} C_DIS
LIN {X -0.108,Y -623.994,Z 1429.370,A 0.000,B 0.000,C 90.000,E1 102.591} C_DIS
LIN {X -0.134,Y -624.088,Z 1429.366,A 0.000,B 0.000,C 90.000,E1 101.827} C_DIS
LIN {X 0.051,Y -623.752,Z 1429.363,A 0.000,B 0.000,C 90.000,E1 101.299} C_DIS
LIN {X 0.115,Y -623.211,Z 1429.360,A 0.000,B 0.000,C 90.000,E1 100.782} C_DIS
LIN {X 0.295,Y -622.298,Z 1429.357,A 0.000,B 0.000,C 90.000,E1 100.254} C_DIS
LIN {X -0.148,Y -621.142,Z 1429.354,A 0.000,B 0.000,C 90.000,E1 99.782} C_DIS
LIN {X -0.090,Y -619.766,Z 1429.351,A 0.000,B 0.000,C 90.000,E1 99.265} C_DIS
LIN {X 0.292,Y -619.007,Z 1429.350,A 0.000,B 0.000,C 90.000,E1 98.973} C_DIS
LIN {X -0.272,Y -617.186,Z 1429.347,A 0.000,B 0.000,C 90.000,E1 98.511} C_DIS
LIN {X -0.232,Y -615.082,Z 1429.344,A 0.000,B 0.000,C 90.000,E1 97.992} C_DIS
LIN {X -0.124,Y -612.531,Z 1429.341,A 0.000,B 0.000,C 90.000,E1 97.466} C_DIS
LIN {X 0.142,Y -608.381,Z 1429.337,A 0.000,B 0.000,C 90.000,E1 96.663} C_DIS
LIN {X 0.121,Y -605.365,Z 1429.334,A 0.000,B 0.000,C 90.000,E1 96.144} C_DIS
LIN {X -0.099,Y -601.017,Z 1429.331,A 0.000,B 0.000,C 90.000,E1 95.511} C_DIS
LIN {X -0.170,Y -596.507,Z 1429.328,A 0.000,B 0.000,C 90.000,E1 94.992} C_DIS
LIN {X -0.160,Y -591.349,Z 1429.325,A 0.000,B 0.000,C 90.000,E1 94.473} C_DIS
LIN {X 0.255,Y -584.074,Z 1429.322,A 0.000,B 0.000,C 90.000,E1 93.841} C_DIS
LIN {X -0.118,Y -577.883,Z 1429.319,A 0.000,B 0.000,C 90.000,E1 93.440} C_DIS
LIN {X -0.038,Y -574.566,Z 1429.318,A 0.000,B 0.000,C 90.000,E1 93.154} C_DIS
LIN {X -0.040,Y -573.373,Z 1429.317,A 0.000,B 0.000,C 90.000,E1 93.037} C_DIS
LIN {X -0.130,Y -572.919,Z 1429.317,A 0.000,B 0.000,C 90.000,E1 92.980} C_DIS
LIN {X 0.008,Y -571.960,Z 1429.315,A 0.000,B 0.000,C 90.000,E1 92.694} C_DIS
LIN {X 0.062,Y -571.656,Z 1429.313,A 0.000,B 0.000,C 90.000,E1 92.407} C_DIS
LIN {X -0.129,Y -571.550,Z 1429.311,A 0.000,B 0.000,C 90.000,E1 91.892} C_DIS
LIN {X 0.127,Y -573.801,Z 1429.295,A 0.000,B 0.000,C 90.000,E1 89.141} C_DIS
LIN {X 0.293,Y -575.039,Z 1429.288,A 0.000,B 0.000,C 90.000,E1 87.764} C_DIS
LIN {X 0.055,Y -576.580,Z 1429.279,A 0.000,B 0.000,C 90.000,E1 86.159} C_DIS
LIN {X -0.271,Y -577.871,Z 1429.271,A 0.000,B 0.000,C 90.000,E1 84.837} C_DIS
LIN {X 0.209,Y -579.502,Z 1429.262,A 0.000,B 0.000,C 90.000,E1 83.166} C_DIS
LIN {X -0.002,Y -580.955,Z 1429.255,A 0.000,B 0.000,C 90.000,E1 81.837} C_DIS
LIN {X 0.241,Y -582.082,Z 1429.249,A 0.000,B 0.000,C 90.000,E1 80.735} C_DIS
LIN {X 0.067,Y -584.085,Z 1429.238,A 0.000,B 0.000,C 90.000,E1 78.870} C_DIS
LIN {X 0.139,Y -585.489,Z 1429.231,A 0.000,B 0.000,C 90.000,E1 77.521} C_DIS
LIN {X 0.155,Y -586.957,Z 1429.220,A 0.000,B 0.000,C 90.000,E1 75.644} C_DIS
LIN {X -0.074,Y -588.171,Z 1429.210,A 0.000,B 0.000,C 90.000,E1 73.795} C_DIS
LIN {X -0.198,Y -588.889,Z 1429.203,A 0.000,B 0.000,C 90.000,E1 72.472} C_DIS
LIN {X -0.073,Y -589.686,Z 1429.194,A 0.000,B 0.000,C 90.000,E1 70.859} C_DIS
LIN {X -0.107,Y -590.652,Z 1429.185,A 0.000,B 0.000,C 90.000,E1 69.263} C_DIS
LIN {X 0.216,Y -591.853,Z 1429.173,A 0.000,B 0.000,C 90.000,E1 67.102} C_DIS
LIN {X 0.013,Y -592.763,Z 1429.166,A 0.000,B 0.000,C 90.000,E1 65.793} C_DIS
LIN {X 0.230,Y -594.426,Z 1429.152,A 0.000,B 0.000,C 90.000,E1 63.384} C_DIS
LIN {X -0.223,Y -595.478,Z 1429.145,A 0.000,B 0.000,C 90.000,E1 62.103} C_DIS
LIN {X 0.253,Y -596.991,Z 1429.135,A 0.000,B 0.000,C 90.000,E1 60.205} C_DIS
LIN {X -0.094,Y -598.180,Z 1429.127,A 0.000,B 0.000,C 90.000,E1 58.918} C_DIS
LIN {X 0.007,Y -599.667,Z 1429.119,A 0.000,B 0.000,C 90.000,E1 57.327} C_DIS
LIN {X 0.185,Y -601.334,Z 1429.108,A 0.000,B 0.000,C 90.000,E1 55.468} C_DIS
LIN {X 0.258,Y -602.918,Z 1429.098,A 0.000,B 0.000,C 90.000,E1 53.623} C_DIS
LIN {X -0.151,Y -603.900,Z 1429.091,A 0.000,B 0.000,C 90.000,E1 52.351} C_DIS
LIN {X 0.196,Y -604.777,Z 1429.083,A 0.000,B 0.000,C 90.000,E1 51.009} C_DIS
LIN {X 0.176,Y -605.516,Z 1429.076,A 0.000,B 0.000,C 90.000,E1 49.703} C_DIS
LIN {X 0.090,Y -605.810,Z 1429.069,A 0.000,B 0.000,C 90.000,E1 48.405} C_DIS
LIN {X 0.034,Y -606.045,Z 1429.059,A 0.000,B 0.000,C 90.000,E1 46.581} C_DIS
LIN {X -0.055,Y -606.112,Z 1429.052,A 0.000,B 0.000,C 90.000,E1 45.283} C_DIS
LIN {X 0.272,Y -605.780,Z 1429.044,A 0.000,B 0.000,C 90.000,E1 43.947} C_DIS
LIN {X -0.115,Y -605.617,Z 1429.041,A 0.000,B 0.000,C 90.000,E1 43.461} C_DIS
LIN {X 0.005,Y -604.619,Z 1429.033,A 0.000,B 0.000,C 90.000,E1 41.881} C_DIS
LIN {X 0.304,Y -604.023,Z 1429.028,A 0.000,B 0.000,C 90.000,E1 41.067} C_DIS
LIN {X 0.009,Y -602.962,Z 1429.023,A 0.000,B 0.000,C 90.000,E1 40.048} C_DIS
LIN {X 0.091,Y -601.819,Z 1429.017,A 0.000,B 0.000,C 90.000,E1 38.991} C_DIS
LIN {X 0.024,Y -600.018,Z 1429.009,A 0.000,B 0.000,C 90.000,E1 37.684} C_DIS
LIN {X 0.281,Y -598.826,Z 1429.005,A 0.000,B 0.000,C 90.000,E1 36.870} C_DIS
LIN {X -0.202,Y -596.341,Z 1428.998,A 0.000,B 0.000,C 90.000,E1 35.598} C_DIS
LIN {X -0.345,Y -594.671,Z 1428.993,A 0.000,B 0.000,C 90.000,E1 34.818} C_DIS
LIN {X -0.017,Y -592.836,Z 1428.989,A 0.000,B 0.000,C 90.000,E1 33.992} C_DIS
LIN {X -0.321,Y -590.120,Z 1428.983,A 0.000,B 0.000,C 90.000,E1 32.959} C_DIS
LIN {X -0.045,Y -587.870,Z 1428.979,A 0.000,B 0.000,C 90.000,E1 32.133} C_DIS
LIN {X 0.019,Y -586.115,Z 1428.976,A 0.000,B 0.000,C 90.000,E1 31.592} C_DIS
LIN {X -0.059,Y -583.280,Z 1428.971,A 0.000,B 0.000,C 90.000,E1 30.797} C_DIS
LIN {X -0.162,Y -580.002,Z 1428.967,A 0.000,B 0.000,C 90.000,E1 30.001} C_DIS
LIN {X 0.130,Y -575.806,Z 1428.961,A 0.000,B 0.000,C 90.000,E1 29.027} C_DIS
LIN {X -0.059,Y -571.692,Z 1428.957,A 0.000,B 0.000,C 90.000,E1 28.231} C_DIS
LIN {X 0.294,Y -567.926,Z 1428.953,A 0.000,B 0.000,C 90.000,E1 27.513} C_DIS
LIN {X -0.243,Y -563.206,Z 1428.948,A 0.000,B 0.000,C 90.000,E1 26.744} C_DIS
LIN {X 0.321,Y -557.084,Z 1428.943,A 0.000,B 0.000,C 90.000,E1 25.720} C_DIS
LIN {X 0.064,Y -550.495,Z 1428.938,A 0.000,B 0.000,C 90.000,E1 24.771} C_DIS
LIN {X 0.097,Y -546.447,Z 1428.935,A 0.000,B 0.000,C 90.000,E1 24.207} C_DIS
LIN {X 0.100,Y -542.100,Z 1428.931,A 0.000,B 0.000,C 90.000,E1 23.643} C_DIS
LIN {X -0.102,Y -535.123,Z 1428.927,A 0.000,B 0.000,C 90.000,E1 22.823} C_DIS
LIN {X 0.009,Y -527.616,Z 1428.922,A 0.000,B 0.000,C 90.000,E1 21.950} C_DIS
LIN {X -0.002,Y -517.432,Z 1428.916,A 0.000,B 0.000,C 90.000,E1 20.844} C_DIS
LIN {X 0.130,Y -506.620,Z 1428.910,A 0.000,B 0.000,C 90.000,E1 19.704} C_DIS
LIN {X 0.256,Y -496.020,Z 1428.904,A 0.000,B 0.000,C 90.000,E1 18.598} C_DIS
LIN {X 0.168,Y -479.682,Z 1428.894,A 0.000,B 0.000,C 90.000,E1 16.913} C_DIS
LIN {X -0.181,Y -466.141,Z 1428.886,A 0.000,B 0.000,C 90.000,E1 15.481} C_DIS
LIN {X 0.200,Y -454.048,Z 1428.878,A 0.000,B 0.000,C 90.000,E1 14.064} C_DIS
LIN {X -0.207,Y -443.321,Z 1428.871,A 0.000,B 0.000,C 90.000,E1 12.883} C_DIS
LIN {X -0.111,Y -432.672,Z 1428.864,A 0.000,B 0.000,C 90.000,E1 11.591} C_DIS
LIN {X -0.100,Y -425.731,Z 1428.860,A 0.000,B 0.000,C 90.000,E1 10.782} C_DIS
LIN {X -0.027,Y -419.838,Z 1428.856,A 0.000,B 0.000,C 90.000,E1 10.141} C_DIS
LIN {X 0.147,Y -415.136,Z 1428.854,A 0.000,B 0.000,C 90.000,E1 9.670} C_DIS
LIN {X 0.053,Y -410.135,Z 1428.852,A 0.000,B 0.000,C 90.000,E1 9.265} C_DIS
LIN {X -0.080,Y -406.312,Z 1428.850,A 0.000,B 0.000,C 90.000,E1 9.029} C_DIS
LIN {X -0.106,Y -403.755,Z 1428.849,A 0.000,B 0.000,C 90.000,E1 8.916} C_DIS
LIN {X 0.005,Y -401.803,Z 1428.849,A 0.000,B 0.000,C 90.000,E1 8.859} C_DIS
LIN {X -0.014,Y -365.371,Z 1428.849,A 0.000,B 0.000,C 90.000,E1 8.859} C_DIS
LIN {X 0.006,Y -361.243,Z 1428.814,A 0.000,B 0.000,C 90.000,E1 2.465} C_DIS
LIN {X -0.069,Y -360.902,Z 1428.801,A 0.000,B 0.000,C 90.000,E1 0.229} C_DIS
LIN {X -0.053,Y -359.426,Z 1428.770,A 0.000,B 0.000,C 90.000,E1 354.546} C_DIS
LIN {X 0.070,Y -358.890,Z 1428.759,A 0.000,B 0.000,C 90.000,E1 352.648} C_DIS
LIN {X -0.020,Y -359.563,Z 1428.726,A 0.000,B 0.000,C 90.000,E1 346.645} C_DIS
LIN {X 0.001,Y -361.801,Z 1428.684,A 0.000,B 0.000,C 90.000,E1 339.135} C_DIS
LIN {X -0.154,Y -362.053,Z 1428.680,A 0.000,B 0.000,C 90.000,E1 338.411} C_DIS
LIN {X 0.189,Y -365.980,Z 1428.643,A 0.000,B 0.000,C 90.000,E1 331.641} C_DIS
LIN {X 0.029,Y -366.387,Z 1428.639,A 0.000,B 0.000,C 90.000,E1 330.923} C_DIS
LIN {X -0.031,Y -371.355,Z 1428.604,A 0.000,B 0.000,C 90.000,E1 324.642} C_DIS
LIN {X -0.043,Y -371.766,Z 1428.602,A 0.000,B 0.000,C 90.000,E1 324.276} C_DIS
LIN {X 0.013,Y -377.358,Z 1428.567,A 0.000,B 0.000,C 90.000,E1 318.038} C_DIS
LIN {X 0.012,Y -378.235,Z 1428.563,A 0.000,B 0.000,C 90.000,E1 317.310} C_DIS
LIN {X 0.002,Y -383.940,Z 1428.531,A 0.000,B 0.000,C 90.000,E1 311.515} C_DIS
LIN {X 0.088,Y -384.893,Z 1428.527,A 0.000,B 0.000,C 90.000,E1 310.782} C_DIS
LIN {X 0.262,Y -390.610,Z 1428.495,A 0.000,B 0.000,C 90.000,E1 305.025} C_DIS
LIN {X 0.106,Y -391.104,Z 1428.493,A 0.000,B 0.000,C 90.000,E1 304.692} C_DIS
LIN {X 0.022,Y -391.648,Z 1428.489,A 0.000,B 0.000,C 90.000,E1 303.992} C_DIS
LIN {X -0.080,Y -396.825,Z 1428.459,A 0.000,B 0.000,C 90.000,E1 298.693} C_DIS
LIN {X -0.210,Y -397.120,Z 1428.457,A 0.000,B 0.000,C 90.000,E1 298.359} C_DIS
LIN {X -0.055,Y -401.597,Z 1428.426,A 0.000,B 0.000,C 90.000,E1 292.717} C_DIS
LIN {X 0.222,Y -404.659,Z 1428.395,A 0.000,B 0.000,C 90.000,E1 287.094} C_DIS
LIN {X -0.079,Y -404.735,Z 1428.391,A 0.000,B 0.000,C 90.000,E1 286.441} C_DIS
LIN {X 0.214,Y -406.099,Z 1428.364,A 0.000,B 0.000,C 90.000,E1 281.535} C_DIS
LIN {X -0.176,Y -406.094,Z 1428.362,A 0.000,B 0.000,C 90.000,E1 281.243} C_DIS
LIN {X -0.097,Y -405.680,Z 1428.333,A 0.000,B 0.000,C 90.000,E1 276.024} C_DIS
LIN {X -0.165,Y -405.058,Z 1428.328,A 0.000,B 0.000,C 90.000,E1 274.992} C_DIS
LIN {X -0.060,Y -403.497,Z 1428.304,A 0.000,B 0.000,C 90.000,E1 270.802} C_DIS
LIN {X -0.092,Y -403.288,Z 1428.302,A 0.000,B 0.000,C 90.000,E1 270.458} C_DIS
LIN {X 0.091,Y -398.931,Z 1428.271,A 0.000,B 0.000,C 90.000,E1 264.837} C_DIS
LIN {X -0.040,Y -393.108,Z 1428.242,A 0.000,B 0.000,C 90.000,E1 259.567} C_DIS
LIN {X -0.079,Y -392.835,Z 1428.240,A 0.000,B 0.000,C 90.000,E1 259.218} C_DIS
LIN {X 0.034,Y -385.993,Z 1428.212,A 0.000,B 0.000,C 90.000,E1 254.212} C_DIS
LIN {X -0.026,Y -385.267,Z 1428.208,A 0.000,B 0.000,C 90.000,E1 253.504} C_DIS
LIN {X -0.004,Y -384.768,Z 1428.206,A 0.000,B 0.000,C 90.000,E1 253.142} C_DIS
LIN {X 0.221,Y -377.973,Z 1428.182,A 0.000,B 0.000,C 90.000,E1 248.773} C_DIS
LIN {X -0.044,Y -376.233,Z 1428.174,A 0.000,B 0.000,C 90.000,E1 247.358} C_DIS
LIN {X 0.057,Y -374.944,Z 1428.170,A 0.000,B 0.000,C 90.000,E1 246.613} C_DIS
LIN {X -0.208,Y -368.417,Z 1428.148,A 0.000,B 0.000,C 90.000,E1 242.615} C_DIS
LIN {X 0.097,Y -366.047,Z 1428.137,A 0.000,B 0.000,C 90.000,E1 240.717} C_DIS
LIN {X 0.004,Y -359.196,Z 1428.115,A 0.000,B 0.000,C 90.000,E1 236.628} C_DIS
LIN {X 0.021,Y -355.842,Z 1428.100,A 0.000,B 0.000,C 90.000,E1 233.989} C_DIS
LIN {X -0.173,Y -348.793,Z 1428.075,A 0.000,B 0.000,C 90.000,E1 229.461} C_DIS
LIN {X -0.097,Y -346.185,Z 1428.062,A 0.000,B 0.000,C 90.000,E1 227.148} C_DIS
LIN {X -0.088,Y -345.065,Z 1428.058,A 0.000,B 0.000,C 90.000,E1 226.377} C_DIS
LIN {X 0.094,Y -338.586,Z 1428.030,A 0.000,B 0.000,C 90.000,E1 221.310} C_DIS
LIN {X 0.094,Y -336.840,Z 1428.019,A 0.000,B 0.000,C 90.000,E1 219.358} C_DIS
LIN {X 0.014,Y -330.861,Z 1427.988,A 0.000,B 0.000,C 90.000,E1 213.865} C_DIS
LIN {X 0.149,Y -329.296,Z 1427.975,A 0.000,B 0.000,C 90.000,E1 211.465} C_DIS
LIN {X -0.154,Y -324.669,Z 1427.942,A 0.000,B 0.000,C 90.000,E1 205.540} C_DIS
LIN {X 0.174,Y -323.837,Z 1427.928,A 0.000,B 0.000,C 90.000,E1 203.078} C_DIS
LIN {X -0.017,Y -321.124,Z 1427.881,A 0.000,B 0.000,C 90.000,E1 194.662} C_DIS
LIN {X 0.138,Y -320.932,Z 1427.877,A 0.000,B 0.000,C 90.000,E1 193.828} C_DIS
LIN {X -0.076,Y -321.562,Z 1427.832,A 0.000,B 0.000,C 90.000,E1 185.796} C_DIS
LIN {X -0.143,Y -324.415,Z 1427.790,A 0.000,B 0.000,C 90.000,E1 178.165} C_DIS
LIN {X -0.141,Y -325.376,Z 1427.783,A 0.000,B 0.000,C 90.000,E1 176.963} C_DIS
LIN {X -0.100,Y -329.112,Z 1427.750,A 0.000,B 0.000,C 90.000,E1 170.971} C_DIS
LIN {X -0.061,Y -329.971,Z 1427.745,A 0.000,B 0.000,C 90.000,E1 170.095} C_DIS
LIN {X -0.081,Y -337.636,Z 1427.745,A 0.000,B 0.000,C 90.000,E1 170.095} C_DIS
LIN {X 0.099,Y -338.651,Z 1427.745,A 0.000,B 0.000,C 90.000,E1 170.038} C_DIS
LIN {X -0.102,Y -341.384,Z 1427.744,A 0.000,B 0.000,C 90.000,E1 169.926} C_DIS
LIN {X 0.095,Y -343.384,Z 1427.743,A 0.000,B 0.000,C 90.000,E1 169.746} C_DIS
LIN {X 0.082,Y -349.376,Z 1427.740,A 0.000,B 0.000,C 90.000,E1 169.218} C_DIS
LIN {X 0.131,Y -353.915,Z 1427.738,A 0.000,B 0.000,C 90.000,E1 168.757} C_DIS
LIN {X 0.041,Y -359.839,Z 1427.734,A 0.000,B 0.000,C 90.000,E1 168.117} C_DIS
LIN {X -0.172,Y -365.697,Z 1427.730,A 0.000,B 0.000,C 90.000,E1 167.465} C_DIS
LIN {X -0.121,Y -378.714,Z 1427.722,A 0.000,B 0.000,C 90.000,E1 165.880} C_DIS
LIN {X -0.077,Y -390.322,Z 1427.715,A 0.000,B 0.000,C 90.000,E1 164.629} C_DIS
LIN {X -0.046,Y -402.608,Z 1427.708,A 0.000,B 0.000,C 90.000,E1 163.449} C_DIS
LIN {X -0.111,Y -419.799,Z 1427.700,A 0.000,B 0.000,C 90.000,E1 161.945} C_DIS
LIN {X -0.218,Y -432.165,Z 1427.694,A 0.000,B 0.000,C 90.000,E1 160.913} C_DIS
LIN {X 0.167,Y -444.600,Z 1427.688,A 0.000,B 0.000,C 90.000,E1 159.826} C_DIS
LIN {X -0.107,Y -456.823,Z 1427.682,A 0.000,B 0.000,C 90.000,E1 158.827} C_DIS
LIN {X 0.104,Y -468.817,Z 1427.677,A 0.000,B 0.000,C 90.000,E1 157.794} C_DIS
LIN {X -0.076,Y -480.503,Z 1427.671,A 0.000,B 0.000,C 90.000,E1 156.794} C_DIS
LIN {X 0.242,Y -487.654,Z 1427.667,A 0.000,B 0.000,C 90.000,E1 156.102} C_DIS
LIN {X -0.169,Y -496.041,Z 1427.663,A 0.000,B 0.000,C 90.000,E1 155.357} C_DIS
LIN {X -0.238,Y -504.143,Z 1427.658,A 0.000,B 0.000,C 90.000,E1 154.537} C_DIS
LIN {X 0.094,Y -508.134,Z 1427.656,A 0.000,B 0.000,C 90.000,E1 154.076} C_DIS
LIN {X 0.152,Y -511.975,Z 1427.654,A 0.000,B 0.000,C 90.000,E1 153.640} C_DIS
LIN {X -0.006,Y -517.874,Z 1427.650,A 0.000,B 0.000,C 90.000,E1 152.922} C_DIS
LIN {X -0.215,Y -522.142,Z 1427.646,A 0.000,B 0.000,C 90.000,E1 152.359} C_DIS
LIN {X 0.005,Y -525.177,Z 1427.644,A 0.000,B 0.000,C 90.000,E1 151.897} C_DIS
LIN {X -0.060,Y -529.472,Z 1427.640,A 0.000,B 0.000,C 90.000,E1 151.179} C_DIS
LIN {X 0.208,Y -531.903,Z 1427.637,A 0.000,B 0.000,C 90.000,E1 150.717} C_DIS
LIN {X 0.204,Y -535.330,Z 1427.634,A 0.000,B 0.000,C 90.000,E1 149.999} C_DIS
LIN {X -0.237,Y -538.351,Z 1427.630,A 0.000,B 0.000,C 90.000,E1 149.331} C_DIS
LIN {X -0.059,Y -540.520,Z 1427.626,A 0.000,B 0.000,C 90.000,E1 148.742} C_DIS
LIN {X -0.327,Y -542.426,Z 1427.623,A 0.000,B 0.000,C 90.000,E1 148.201} C_DIS
LIN {X -0.102,Y -544.953,Z 1427.619,A 0.000,B 0.000,C 90.000,E1 147.327} C_DIS
LIN {X -0.307,Y -547.241,Z 1427.614,A 0.000,B 0.000,C 90.000,E1 146.501} C_DIS
LIN {X 0.012,Y -549.835,Z 1427.608,A 0.000,B 0.000,C 90.000,E1 145.341} C_DIS
LIN {X 0.231,Y -552.030,Z 1427.601,A 0.000,B 0.000,C 90.000,E1 144.196} C_DIS
LIN {X 0.029,Y -552.919,Z 1427.598,A 0.000,B 0.000,C 90.000,E1 143.657} C_DIS
LIN {X -0.146,Y -554.399,Z 1427.592,A 0.000,B 0.000,C 90.000,E1 142.557} C_DIS
LIN {X 0.068,Y -555.372,Z 1427.587,A 0.000,B 0.000,C 90.000,E1 141.698} C_DIS
LIN {X 0.006,Y -556.716,Z 1427.580,A 0.000,B 0.000,C 90.000,E1 140.312} C_DIS
LIN {X -0.105,Y -557.786,Z 1427.572,A 0.000,B 0.000,C 90.000,E1 138.933} C_DIS
LIN {X 0.150,Y -558.574,Z 1427.566,A 0.000,B 0.000,C 90.000,E1 137.796} C_DIS
LIN {X 0.120,Y -559.554,Z 1427.556,A 0.000,B 0.000,C 90.000,E1 136.134} C_DIS
LIN {X -0.022,Y -560.062,Z 1427.550,A 0.000,B 0.000,C 90.000,E1 135.040} C_DIS
LIN {X -0.156,Y -560.427,Z 1427.544,A 0.000,B 0.000,C 90.000,E1 133.947} C_DIS
LIN {X 0.183,Y -560.791,Z 1427.536,A 0.000,B 0.000,C 90.000,E1 132.528} C_DIS
LIN {X 0.062,Y -560.877,Z 1427.530,A 0.000,B 0.000,C 90.000,E1 131.434} C_DIS
LIN {X 0.112,Y -560.997,Z 1427.521,A 0.000,B 0.000,C 90.000,E1 129.769} C_DIS
LIN {X 0.146,Y -561.079,Z 1427.513,A 0.000,B 0.000,C 90.000,E1 128.382} C_DIS
LIN {X -0.057,Y -561.087,Z 1427.504,A 0.000,B 0.000,C 90.000,E1 126.744} C_DIS
LIN {X -0.160,Y -560.945,Z 1427.493,A 0.000,B 0.000,C 90.000,E1 124.818} C_DIS
LIN {X -0.230,Y -560.717,Z 1427.484,A 0.000,B 0.000,C 90.000,E1 123.166} C_DIS
LIN {X -0.083,Y -560.640,Z 1427.461,A 0.000,B 0.000,C 90.000,E1 118.999} C_DIS
LIN {X -0.179,Y -561.382,Z 1427.449,A 0.000,B 0.000,C 90.000,E1 116.796} C_DIS
LIN {X -0.161,Y -561.927,Z 1427.441,A 0.000,B 0.000,C 90.000,E1 115.412} C_DIS
LIN {X 0.074,Y -562.244,Z 1427.435,A 0.000,B 0.000,C 90.000,E1 114.283} C_DIS
LIN {X -0.200,Y -562.535,Z 1427.429,A 0.000,B 0.000,C 90.000,E1 113.206} C_DIS
LIN {X 0.238,Y -563.111,Z 1427.424,A 0.000,B 0.000,C 90.000,E1 112.333} C_DIS
LIN {X 0.037,Y -563.426,Z 1427.423,A 0.000,B 0.000,C 90.000,E1 112.078} C_DIS
LIN {X 0.165,Y -564.176,Z 1427.421,A 0.000,B 0.000,C 90.000,E1 111.663} C_DIS
LIN {X 0.065,Y -564.904,Z 1427.420,A 0.000,B 0.000,C 90.000,E1 111.535} C_DIS
LIN {X 0.033,Y -566.154,Z 1427.419,A 0.000,B 0.000,C 90.000,E1 111.354} C_DIS
LIN {X -0.166,Y -569.688,Z 1427.417,A 0.000,B 0.000,C 90.000,E1 111.099} C_DIS
LIN {X 0.247,Y -580.229,Z 1427.414,A 0.000,B 0.000,C 90.000,E1 110.482} C_DIS
LIN {X 0.128,Y -585.852,Z 1427.412,A 0.000,B 0.000,C 90.000,E1 110.120} C_DIS
LIN {X 0.023,Y -591.406,Z 1427.410,A 0.000,B 0.000,C 90.000,E1 109.704} C_DIS
LIN {X -0.276,Y -596.721,Z 1427.407,A 0.000,B 0.000,C 90.000,E1 109.268} C_DIS
LIN {X -0.252,Y -601.754,Z 1427.404,A 0.000,B 0.000,C 90.000,E1 108.779} C_DIS
LIN {X 0.079,Y -606.435,Z 1427.401,A 0.000,B 0.000,C 90.000,E1 108.236} C_DIS
LIN {X 0.307,Y -610.818,Z 1427.399,A 0.000,B 0.000,C 90.000,E1 107.692} C_DIS
LIN {X 0.014,Y -613.536,Z 1427.396,A 0.000,B 0.000,C 90.000,E1 107.330} C_DIS
LIN {X 0.319,Y -616.171,Z 1427.394,A 0.000,B 0.000,C 90.000,E1 106.913} C_DIS
LIN {X 0.211,Y -620.196,Z 1427.390,A 0.000,B 0.000,C 90.000,E1 106.150} C_DIS
LIN {X -0.067,Y -621.893,Z 1427.387,A 0.000,B 0.000,C 90.000,E1 105.662} C_DIS
LIN {X -0.287,Y -622.639,Z 1427.386,A 0.000,B 0.000,C 90.000,E1 105.426} C_DIS
LIN {X -0.117,Y -623.772,Z 1427.383,A 0.000,B 0.000,C 90.000,E1 104.898} C_DIS
LIN {X 0.201,Y -625.665,Z 1427.376,A 0.000,B 0.000,C 90.000,E1 103.592} C_DIS
LIN {X -0.212,Y -626.268,Z 1427.373,A 0.000,B 0.000,C 90.000,E1 103.119} C_DIS
LIN {X -0.214,Y -626.645,Z 1427.369,A 0.000,B 0.000,C 90.000,E1 102.355} C_DIS
LIN {X -0.010,Y -626.677,Z 1427.366,A 0.000,B 0.000,C 90.000,E1 101.827} C_DIS
LIN {X -0.134,Y -626.123,Z 1427.361,A 0.000,B 0.000,C 90.000,E1 101.074} C_DIS
LIN {X 0.068,Y -625.442,Z 1427.359,A 0.000,B 0.000,C 90.000,E1 100.546} C_DIS
LIN {X 0.261,Y -624.466,Z 1427.356,A 0.000,B 0.000,C 90.000,E1 100.018} C_DIS
LIN {X -0.275,Y -623.211,Z 1427.353,A 0.000,B 0.000,C 90.000,E1 99.557} C_DIS
LIN {X -0.100,Y -621.684,Z 1427.350,A 0.000,B 0.000,C 90.000,E1 99.029} C_DIS
LIN {X -0.035,Y -619.882,Z 1427.347,A 0.000,B 0.000,C 90.000,E1 98.511} C_DIS
LIN {X 0.022,Y -617.820,Z 1427.344,A 0.000,B 0.000,C 90.000,E1 97.992} C_DIS
LIN {X -0.181,Y -614.217,Z 1427.340,A 0.000,B 0.000,C 90.000,E1 97.239} C_DIS
LIN {X 0.008,Y -609.151,Z 1427.335,A 0.000,B 0.000,C 90.000,E1 96.315} C_DIS
LIN {X -0.182,Y -605.130,Z 1427.332,A 0.000,B 0.000,C 90.000,E1 95.682} C_DIS
LIN {X 0.246,Y -604.270,Z 1427.331,A 0.000,B 0.000,C 90.000,E1 95.511} C_DIS
LIN {X 0.016,Y -598.818,Z 1427.327,A 0.000,B 0.000,C 90.000,E1 94.878} C_DIS
LIN {X 0.051,Y -593.663,Z 1427.324,A 0.000,B 0.000,C 90.000,E1 94.359} C_DIS
LIN {X -0.214,Y -590.824,Z 1427.323,A 0.000,B 0.000,C 90.000,E1 94.131} C_DIS
LIN {X -0.273,Y -584.989,Z 1427.320,A 0.000,B 0.000,C 90.000,E1 93.669} C_DIS
LIN {X 0.218,Y -575.943,Z 1427.317,A 0.000,B 0.000,C 90.000,E1 92.980} C_DIS
LIN {X -0.166,Y -573.661,Z 1427.316,A 0.000,B 0.000,C 90.000,E1 92.808} C_DIS
LIN {X -0.225,Y -573.115,Z 1427.315,A 0.000,B 0.000,C 90.000,E1 92.751} C_DIS
LIN {X 0.115,Y -572.162,Z 1427.314,A 0.000,B 0.000,C 90.000,E1 92.465} C_DIS
LIN {X 0.060,Y -571.719,Z 1427.312,A 0.000,B 0.000,C 90.000,E1 92.064} C_DIS
LIN {X 0.154,Y -571.905,Z 1427.307,A 0.000,B 0.000,C 90.000,E1 91.318} C_DIS
LIN {X -0.019,Y -573.515,Z 1427.297,A 0.000,B 0.000,C 90.000,E1 89.427} C_DIS
LIN {X 0.143,Y -574.801,Z 1427.289,A 0.000,B 0.000,C 90.000,E1 88.051} C_DIS
LIN {X -0.096,Y -576.316,Z 1427.280,A 0.000,B 0.000,C 90.000,E1 86.445} C_DIS
LIN {X 0.154,Y -577.622,Z 1427.273,A 0.000,B 0.000,C 90.000,E1 85.065} C_DIS
LIN {X 0.060,Y -579.223,Z 1427.264,A 0.000,B 0.000,C 90.000,E1 83.451} C_DIS
LIN {X -0.006,Y -580.987,Z 1427.255,A 0.000,B 0.000,C 90.000,E1 81.837} C_DIS
LIN {X -0.105,Y -582.404,Z 1427.247,A 0.000,B 0.000,C 90.000,E1 80.500} C_DIS
LIN {X 0.064,Y -584.133,Z 1427.238,A 0.000,B 0.000,C 90.000,E1 78.870} C_DIS
LIN {X 0.137,Y -585.534,Z 1427.231,A 0.000,B 0.000,C 90.000,E1 77.521} C_DIS
LIN {X 0.155,Y -586.985,Z 1427.220,A 0.000,B 0.000,C 90.000,E1 75.644} C_DIS
LIN {X 0.084,Y -588.036,Z 1427.211,A 0.000,B 0.000,C 90.000,E1 74.047} C_DIS
LIN {X 0.046,Y -589.079,Z 1427.201,A 0.000,B 0.000,C 90.000,E1 72.181} C_DIS
LIN {X -0.070,Y -589.753,Z 1427.194,A 0.000,B 0.000,C 90.000,E1 70.859} C_DIS
LIN {X -0.102,Y -590.696,Z 1427.185,A 0.000,B 0.000,C 90.000,E1 69.263} C_DIS
LIN {X -0.111,Y -591.553,Z 1427.176,A 0.000,B 0.000,C 90.000,E1 67.667} C_DIS
LIN {X 0.221,Y -592.475,Z 1427.169,A 0.000,B 0.000,C 90.000,E1 66.305} C_DIS
LIN {X -0.018,Y -593.846,Z 1427.157,A 0.000,B 0.000,C 90.000,E1 64.204} C_DIS
LIN {X -0.034,Y -595.154,Z 1427.148,A 0.000,B 0.000,C 90.000,E1 62.615} C_DIS
LIN {X -0.284,Y -596.403,Z 1427.139,A 0.000,B 0.000,C 90.000,E1 61.051} C_DIS
LIN {X -0.301,Y -598.018,Z 1427.129,A 0.000,B 0.000,C 90.000,E1 59.203} C_DIS
LIN {X 0.023,Y -599.758,Z 1427.119,A 0.000,B 0.000,C 90.000,E1 57.327} C_DIS
LIN {X -0.041,Y -601.178,Z 1427.110,A 0.000,B 0.000,C 90.000,E1 55.754} C_DIS
LIN {X 0.109,Y -602.092,Z 1427.104,A 0.000,B 0.000,C 90.000,E1 54.689} C_DIS
LIN {X -0.311,Y -603.202,Z 1427.097,A 0.000,B 0.000,C 90.000,E1 53.417} C_DIS
LIN {X 0.127,Y -604.164,Z 1427.089,A 0.000,B 0.000,C 90.000,E1 52.065} C_DIS
LIN {X -0.372,Y -605.052,Z 1427.082,A 0.000,B 0.000,C 90.000,E1 50.803} C_DIS
LIN {X -0.001,Y -605.720,Z 1427.075,A 0.000,B 0.000,C 90.000,E1 49.461} C_DIS
LIN {X -0.081,Y -605.948,Z 1427.068,A 0.000,B 0.000,C 90.000,E1 48.162} C_DIS
LIN {X 0.311,Y -606.182,Z 1427.057,A 0.000,B 0.000,C 90.000,E1 46.296} C_DIS
LIN {X 0.212,Y -606.181,Z 1427.050,A 0.000,B 0.000,C 90.000,E1 45.000} C_DIS
LIN {X 0.304,Y -605.868,Z 1427.044,A 0.000,B 0.000,C 90.000,E1 43.947} C_DIS
LIN {X -0.081,Y -605.709,Z 1427.042,A 0.000,B 0.000,C 90.000,E1 43.461} C_DIS
LIN {X -0.167,Y -604.930,Z 1427.034,A 0.000,B 0.000,C 90.000,E1 42.162} C_DIS
LIN {X 0.342,Y -604.162,Z 1427.028,A 0.000,B 0.000,C 90.000,E1 41.067} C_DIS
LIN {X 0.048,Y -603.141,Z 1427.023,A 0.000,B 0.000,C 90.000,E1 40.048} C_DIS
LIN {X 0.133,Y -601.964,Z 1427.017,A 0.000,B 0.000,C 90.000,E1 38.991} C_DIS
LIN {X 0.189,Y -600.552,Z 1427.011,A 0.000,B 0.000,C 90.000,E1 37.935} C_DIS
LIN {X 0.327,Y -599.013,Z 1427.005,A 0.000,B 0.000,C 90.000,E1 36.870} C_DIS
LIN {X -0.038,Y -597.091,Z 1426.999,A 0.000,B 0.000,C 90.000,E1 35.851} C_DIS
LIN {X -0.295,Y -594.891,Z 1426.993,A 0.000,B 0.000,C 90.000,E1 34.818} C_DIS
LIN {X 0.035,Y -593.081,Z 1426.989,A 0.000,B 0.000,C 90.000,E1 33.992} C_DIS
LIN {X -0.266,Y -590.353,Z 1426.983,A 0.000,B 0.000,C 90.000,E1 32.959} C_DIS
LIN {X 0.012,Y -588.102,Z 1426.979,A 0.000,B 0.000,C 90.000,E1 32.133} C_DIS
LIN {X 0.079,Y -586.392,Z 1426.976,A 0.000,B 0.000,C 90.000,E1 31.592} C_DIS
LIN {X 0.004,Y -583.589,Z 1426.971,A 0.000,B 0.000,C 90.000,E1 30.797} C_DIS
LIN {X -0.098,Y -580.338,Z 1426.967,A 0.000,B 0.000,C 90.000,E1 30.001} C_DIS
LIN {X -0.306,Y -576.134,Z 1426.961,A 0.000,B 0.000,C 90.000,E1 29.077} C_DIS
LIN {X 0.013,Y -572.035,Z 1426.957,A 0.000,B 0.000,C 90.000,E1 28.231} C_DIS
LIN {X 0.282,Y -567.546,Z 1426.952,A 0.000,B 0.000,C 90.000,E1 27.385} C_DIS
LIN {X -0.260,Y -562.757,Z 1426.948,A 0.000,B 0.000,C 90.000,E1 26.616} C_DIS
LIN {X -0.098,Y -557.521,Z 1426.943,A 0.000,B 0.000,C 90.000,E1 25.771} C_DIS
LIN {X 0.036,Y -549.988,Z 1426.937,A 0.000,B 0.000,C 90.000,E1 24.643} C_DIS
LIN {X -0.057,Y -544.812,Z 1426.933,A 0.000,B 0.000,C 90.000,E1 23.951} C_DIS
LIN {X -0.066,Y -540.339,Z 1426.930,A 0.000,B 0.000,C 90.000,E1 23.387} C_DIS
LIN {X 0.246,Y -534.326,Z 1426.926,A 0.000,B 0.000,C 90.000,E1 22.642} C_DIS
LIN {X 0.152,Y -526.794,Z 1426.921,A 0.000,B 0.000,C 90.000,E1 21.791} C_DIS
LIN {X -0.146,Y -517.800,Z 1426.916,A 0.000,B 0.000,C 90.000,E1 20.844} C_DIS
LIN {X 0.139,Y -507.136,Z 1426.910,A 0.000,B 0.000,C 90.000,E1 19.704} C_DIS
LIN {X -0.048,Y -496.152,Z 1426.903,A 0.000,B 0.000,C 90.000,E1 18.598} C_DIS
LIN {X 0.187,Y -479.656,Z 1426.894,A 0.000,B 0.000,C 90.000,E1 16.858} C_DIS
LIN {X -0.024,Y -466.246,Z 1426.886,A 0.000,B 0.000,C 90.000,E1 15.426} C_DIS
LIN {X 0.002,Y -454.215,Z 1426.878,A 0.000,B 0.000,C 90.000,E1 14.064} C_DIS
LIN {X 0.088,Y -438.160,Z 1426.868,A 0.000,B 0.000,C 90.000,E1 12.187} C_DIS
LIN {X -0.075,Y -423.467,Z 1426.858,A 0.000,B 0.000,C 90.000,E1 10.433} C_DIS
LIN {X 0.149,Y -419.198,Z 1426.855,A 0.000,B 0.000,C 90.000,E1 9.905} C_DIS
LIN {X 0.186,Y -413.255,Z 1426.852,A 0.000,B 0.000,C 90.000,E1 9.265} C_DIS
LIN {X -0.185,Y -408.550,Z 1426.849,A 0.000,B 0.000,C 90.000,E1 8.859} C_DIS
LIN {X -0.137,Y -405.210,Z 1426.848,A 0.000,B 0.000,C 90.000,E1 8.568} C_DIS
LIN {X 0.058,Y -401.619,Z 1426.846,A 0.000,B 0.000,C 90.000,E1 8.276} C_DIS
LIN {X 0.040,Y -399.641,Z 1426.845,A 0.000,B 0.000,C 90.000,E1 8.163} C_DIS
LIN {X 0.022,Y -396.077,Z 1426.845,A 0.000,B 0.000,C 90.000,E1 8.049} C_DIS
LIN {X -0.010,Y -364.584,Z 1426.845,A 0.000,B 0.000,C 90.000,E1 8.049} C_DIS
LIN {X 0.019,Y -360.912,Z 1426.803,A 0.000,B 0.000,C 90.000,E1 0.458} C_DIS
LIN {X 0.137,Y -360.684,Z 1426.799,A 0.000,B 0.000,C 90.000,E1 359.771} C_DIS
LIN {X -0.053,Y -359.426,Z 1426.770,A 0.000,B 0.000,C 90.000,E1 354.546} C_DIS
LIN {X 0.070,Y -358.890,Z 1426.759,A 0.000,B 0.000,C 90.000,E1 352.648} C_DIS
LIN {X -0.020,Y -359.563,Z 1426.726,A 0.000,B 0.000,C 90.000,E1 346.645} C_DIS
LIN {X 0.001,Y -361.801,Z 1426.684,A 0.000,B 0.000,C 90.000,E1 339.135} C_DIS
LIN {X -0.154,Y -362.053,Z 1426.680,A 0.000,B 0.000,C 90.000,E1 338.411} C_DIS
LIN {X 0.189,Y -365.980,Z 1426.643,A 0.000,B 0.000,C 90.000,E1 331.641} C_DIS
LIN {X 0.029,Y -366.387,Z 1426.639,A 0.000,B 0.000,C 90.000,E1 330.923} C_DIS
LIN {X -0.031,Y -371.355,Z 1426.604,A 0.000,B 0.000,C 90.000,E1 324.642} C_DIS
LIN {X -0.043,Y -371.766,Z 1426.602,A 0.000,B 0.000,C 90.000,E1 324.276} C_DIS
LIN {X 0.013,Y -377.358,Z 1426.567,A 0.000,B 0.000,C 90.000,E1 318.038} C_DIS
LIN {X 0.012,Y -378.235,Z 1426.563,A 0.000,B 0.000,C 90.000,E1 317.310} C_DIS
LIN {X 0.002,Y -383.940,Z 1426.531,A 0.000,B 0.000,C 90.000,E1 311.515} C_DIS
LIN {X 0.088,Y -384.893,Z 1426.527,A 0.000,B 0.000,C 90.000,E1 310.782} C_DIS
LIN {X 0.262,Y -390.610,Z 1426.495,A 0.000,B 0.000,C 90.000,E1 305.025} C_DIS
LIN {X 0.106,Y -391.104,Z 1426.493,A 0.000,B 0.000,C 90.000,E1 304.692} C_DIS
LIN {X 0.022,Y -391.648,Z 1426.489,A 0.000,B 0.000,C 90.000,E1 303.992} C_DIS
LIN {X -0.080,Y -396.825,Z 1426.459,A 0.000,B 0.000,C 90.000,E1 298.693} C_DIS
LIN {X -0.210,Y -397.120,Z 1426.457,A 0.000,B 0.000,C 90.000,E1 298.359} C_DIS
LIN {X -0.055,Y -401.597,Z 1426.426,A 0.000,B 0.000,C 90.000,E1 292.717} C_DIS
LIN {X 0.222,Y -404.659,Z 1426.395,A 0.000,B 0.000,C 90.000,E1 287.094} C_DIS
LIN {X -0.079,Y -404.735,Z 1426.391,A 0.000,B 0.000,C 90.000,E1 286.441} C_DIS
LIN {X 0.214,Y -406.099,Z 1426.364,A 0.000,B 0.000,C 90.000,E1 281.535} C_DIS
LIN {X -0.176,Y -406.094,Z 1426.362,A 0.000,B 0.000,C 90.000,E1 281.243} C_DIS
LIN {X -0.097,Y -405.680,Z 1426.333,A 0.000,B 0.000,C 90.000,E1 276.024} C_DIS
LIN {X -0.165,Y -405.058,Z 1426.328,A 0.000,B 0.000,C 90.000,E1 274.992} C_DIS
LIN {X -0.060,Y -403.497,Z 1426.304,A 0.000,B 0.000,C 90.000,E1 270.802} C_DIS
LIN {X -0.092,Y -403.288,Z 1426.302,A 0.000,B 0.000,C 90.000,E1 270.458} C_DIS
LIN {X 0.091,Y -398.931,Z 1426.271,A 0.000,B 0.000,C 90.000,E1 264.837} C_DIS
LIN {X -0.040,Y -393.108,Z 1426.242,A 0.000,B 0.000,C 90.000,E1 259.567} C_DIS
LIN {X -0.079,Y -392.835,Z 1426.240,A 0.000,B 0.000,C 90.000,E1 259.218} C_DIS
LIN {X 0.034,Y -385.993,Z 1426.212,A 0.000,B 0.000,C 90.000,E1 254.212} C_DIS
LIN {X -0.026,Y -385.267,Z 1426.208,A 0.000,B 0.000,C 90.000,E1 253.504} C_DIS
LIN {X -0.004,Y -384.768,Z 1426.206,A 0.000,B 0.000,C 90.000,E1 253.142} C_DIS
LIN {X 0.221,Y -377.973,Z 1426.182,A 0.000,B 0.000,C 90.000,E1 248.773} C_DIS
LIN {X -0.044,Y -376.233,Z 1426.174,A 0.000,B 0.000,C 90.000,E1 247.358} C_DIS
LIN {X 0.057,Y -374.944,Z 1426.170,A 0.000,B 0.000,C 90.000,E1 246.613} C_DIS
LIN {X -0.208,Y -368.417,Z 1426.148,A 0.000,B 0.000,C 90.000,E1 242.615} C_DIS
LIN {X 0.097,Y -366.047,Z 1426.137,A 0.000,B 0.000,C 90.000,E1 240.717} C_DIS
LIN {X 0.004,Y -359.196,Z 1426.115,A 0.000,B 0.000,C 90.000,E1 236.628} C_DIS
LIN {X 0.021,Y -355.842,Z 1426.100,A 0.000,B 0.000,C 90.000,E1 233.989} C_DIS
LIN {X -0.173,Y -348.793,Z 1426.075,A 0.000,B 0.000,C 90.000,E1 229.461} C_DIS
LIN {X -0.097,Y -346.185,Z 1426.062,A 0.000,B 0.000,C 90.000,E1 227.148} C_DIS
LIN {X -0.088,Y -345.065,Z 1426.058,A 0.000,B 0.000,C 90.000,E1 226.377} C_DIS
LIN {X 0.094,Y -338.586,Z 1426.030,A 0.000,B 0.000,C 90.000,E1 221.310} C_DIS
LIN {X 0.094,Y -336.840,Z 1426.019,A 0.000,B 0.000,C 90.000,E1 219.358} C_DIS
LIN {X 0.014,Y -330.861,Z 1425.988,A 0.000,B 0.000,C 90.000,E1 213.865} C_DIS
LIN {X 0.149,Y -329.296,Z 1425.975,A 0.000,B 0.000,C 90.000,E1 211.465} C_DIS
LIN {X -0.154,Y -324.669,Z 1425.942,A 0.000,B 0.000,C 90.000,E1 205.540} C_DIS
LIN {X 0.174,Y -323.837,Z 1425.928,A 0.000,B 0.000,C 90.000,E1 203.078} C_DIS
LIN {X -0.017,Y -321.124,Z 1425.881,A 0.000,B 0.000,C 90.000,E1 194.662} C_DIS
LIN {X 0.138,Y -320.932,Z 1425.877,A 0.000,B 0.000,C 90.000,E1 193.828} C_DIS
LIN {X -0.076,Y -321.562,Z 1425.832,A 0.000,B 0.000,C 90.000,E1 185.796} C_DIS
LIN {X -0.143,Y -324.415,Z 1425.790,A 0.000,B 0.000,C 90.000,E1 178.165} C_DIS
LIN {X -0.141,Y -325.376,Z 1425.783,A 0.000,B 0.000,C 90.000,E1 176.963} C_DIS
LIN {X -0.036,Y -328.996,Z 1425.750,A 0.000,B 0.000,C 90.000,E1 171.084} C_DIS
LIN {X -0.055,Y -333.160,Z 1425.750,A 0.000,B 0.000,C 90.000,E1 171.084} C_DIS
LIN {X 0.148,Y -333.986,Z 1425.750,A 0.000,B 0.000,C 90.000,E1 171.027} C_DIS
LIN {X -0.103,Y -335.717,Z 1425.750,A 0.000,B 0.000,C 90.000,E1 170.971} C_DIS
LIN {X 0.137,Y -337.994,Z 1425.749,A 0.000,B 0.000,C 90.000,E1 170.735} C_DIS
LIN {X -0.059,Y -343.569,Z 1425.745,A 0.000,B 0.000,C 90.000,E1 170.151} C_DIS
LIN {X -0.010,Y -353.616,Z 1425.739,A 0.000,B 0.000,C 90.000,E1 168.993} C_DIS
LIN {X -0.050,Y -360.787,Z 1425.734,A 0.000,B 0.000,C 90.000,E1 168.105} C_DIS
LIN {X 0.143,Y -373.621,Z 1425.725,A 0.000,B 0.000,C 90.000,E1 166.464} C_DIS
LIN {X 0.063,Y -383.594,Z 1425.719,A 0.000,B 0.000,C 90.000,E1 165.338} C_DIS
LIN {X -0.020,Y -395.837,Z 1425.712,A 0.000,B 0.000,C 90.000,E1 164.102} C_DIS
LIN {X 0.130,Y -416.171,Z 1425.702,A 0.000,B 0.000,C 90.000,E1 162.253} C_DIS
LIN {X -0.098,Y -428.688,Z 1425.696,A 0.000,B 0.000,C 90.000,E1 161.221} C_DIS
LIN {X -0.051,Y -444.090,Z 1425.688,A 0.000,B 0.000,C 90.000,E1 159.934} C_DIS
LIN {X 0.040,Y -457.686,Z 1425.682,A 0.000,B 0.000,C 90.000,E1 158.773} C_DIS
LIN {X 0.224,Y -468.450,Z 1425.677,A 0.000,B 0.000,C 90.000,E1 157.847} C_DIS
LIN {X -0.120,Y -478.879,Z 1425.672,A 0.000,B 0.000,C 90.000,E1 156.975} C_DIS
LIN {X -0.056,Y -487.595,Z 1425.668,A 0.000,B 0.000,C 90.000,E1 156.177} C_DIS
LIN {X -0.171,Y -494.521,Z 1425.664,A 0.000,B 0.000,C 90.000,E1 155.537} C_DIS
LIN {X -0.024,Y -500.020,Z 1425.661,A 0.000,B 0.000,C 90.000,E1 154.973} C_DIS
LIN {X -0.197,Y -508.074,Z 1425.656,A 0.000,B 0.000,C 90.000,E1 154.152} C_DIS
LIN {X -0.103,Y -513.127,Z 1425.653,A 0.000,B 0.000,C 90.000,E1 153.563} C_DIS
LIN {X -0.143,Y -516.757,Z 1425.651,A 0.000,B 0.000,C 90.000,E1 153.127} C_DIS
LIN {X 0.177,Y -522.118,Z 1425.647,A 0.000,B 0.000,C 90.000,E1 152.359} C_DIS
LIN {X -0.065,Y -525.215,Z 1425.644,A 0.000,B 0.000,C 90.000,E1 151.948} C_DIS
LIN {X 0.337,Y -529.523,Z 1425.640,A 0.000,B 0.000,C 90.000,E1 151.179} C_DIS
LIN {X -0.116,Y -531.957,Z 1425.638,A 0.000,B 0.000,C 90.000,E1 150.795} C_DIS
LIN {X -0.125,Y -535.417,Z 1425.634,A 0.000,B 0.000,C 90.000,E1 150.078} C_DIS
LIN {X 0.168,Y -538.420,Z 1425.630,A 0.000,B 0.000,C 90.000,E1 149.331} C_DIS
LIN {X -0.113,Y -540.604,Z 1425.627,A 0.000,B 0.000,C 90.000,E1 148.791} C_DIS
LIN {X 0.081,Y -542.506,Z 1425.623,A 0.000,B 0.000,C 90.000,E1 148.201} C_DIS
LIN {X -0.149,Y -545.050,Z 1425.619,A 0.000,B 0.000,C 90.000,E1 147.375} C_DIS
LIN {X 0.072,Y -546.643,Z 1425.616,A 0.000,B 0.000,C 90.000,E1 146.786} C_DIS
LIN {X -0.072,Y -549.325,Z 1425.609,A 0.000,B 0.000,C 90.000,E1 145.674} C_DIS
LIN {X 0.085,Y -551.063,Z 1425.605,A 0.000,B 0.000,C 90.000,E1 144.815} C_DIS
LIN {X -0.057,Y -552.601,Z 1425.600,A 0.000,B 0.000,C 90.000,E1 143.989} C_DIS
LIN {X 0.207,Y -554.065,Z 1425.594,A 0.000,B 0.000,C 90.000,E1 142.844} C_DIS
LIN {X 0.057,Y -555.383,Z 1425.588,A 0.000,B 0.000,C 90.000,E1 141.743} C_DIS
LIN {X 0.003,Y -556.699,Z 1425.580,A 0.000,B 0.000,C 90.000,E1 140.356} C_DIS
LIN {X 0.245,Y -557.578,Z 1425.574,A 0.000,B 0.000,C 90.000,E1 139.218} C_DIS
LIN {X -0.287,Y -558.357,Z 1425.568,A 0.000,B 0.000,C 90.000,E1 138.162} C_DIS
LIN {X 0.090,Y -559.361,Z 1425.558,A 0.000,B 0.000,C 90.000,E1 136.458} C_DIS
LIN {X -0.053,Y -559.921,Z 1425.552,A 0.000,B 0.000,C 90.000,E1 135.364} C_DIS
LIN {X -0.191,Y -560.297,Z 1425.546,A 0.000,B 0.000,C 90.000,E1 134.271} C_DIS
LIN {X 0.148,Y -560.672,Z 1425.538,A 0.000,B 0.000,C 90.000,E1 132.852} C_DIS
LIN {X 0.030,Y -560.829,Z 1425.532,A 0.000,B 0.000,C 90.000,E1 131.757} C_DIS
LIN {X 0.177,Y -560.947,Z 1425.521,A 0.000,B 0.000,C 90.000,E1 129.806} C_DIS
LIN {X -0.219,Y -561.030,Z 1425.514,A 0.000,B 0.000,C 90.000,E1 128.463} C_DIS
LIN {X -0.084,Y -561.065,Z 1425.504,A 0.000,B 0.000,C 90.000,E1 126.790} C_DIS
LIN {X 0.166,Y -560.957,Z 1425.495,A 0.000,B 0.000,C 90.000,E1 125.105} C_DIS
LIN {X 0.227,Y -560.841,Z 1425.489,A 0.000,B 0.000,C 90.000,E1 123.992} C_DIS
LIN {X 0.067,Y -560.591,Z 1425.481,A 0.000,B 0.000,C 90.000,E1 122.625} C_DIS
LIN {X -0.066,Y -560.878,Z 1425.458,A 0.000,B 0.000,C 90.000,E1 118.487} C_DIS
LIN {X -0.151,Y -561.727,Z 1425.446,A 0.000,B 0.000,C 90.000,E1 116.283} C_DIS
LIN {X -0.126,Y -562.202,Z 1425.438,A 0.000,B 0.000,C 90.000,E1 114.899} C_DIS
LIN {X 0.231,Y -562.650,Z 1425.429,A 0.000,B 0.000,C 90.000,E1 113.206} C_DIS
LIN {X 0.150,Y -563.329,Z 1425.425,A 0.000,B 0.000,C 90.000,E1 112.386} C_DIS
LIN {X -0.262,Y -563.825,Z 1425.423,A 0.000,B 0.000,C 90.000,E1 112.153} C_DIS
LIN {X 0.161,Y -564.255,Z 1425.422,A 0.000,B 0.000,C 90.000,E1 111.972} C_DIS
LIN {X 0.062,Y -564.853,Z 1425.421,A 0.000,B 0.000,C 90.000,E1 111.844} C_DIS
LIN {X 0.183,Y -566.910,Z 1425.420,A 0.000,B 0.000,C 90.000,E1 111.535} C_DIS
LIN {X -0.157,Y -570.434,Z 1425.418,A 0.000,B 0.000,C 90.000,E1 111.334} C_DIS
LIN {X -0.088,Y -580.824,Z 1425.416,A 0.000,B 0.000,C 90.000,E1 110.791} C_DIS
LIN {X -0.039,Y -586.583,Z 1425.414,A 0.000,B 0.000,C 90.000,E1 110.429} C_DIS
LIN {X 0.126,Y -591.881,Z 1425.411,A 0.000,B 0.000,C 90.000,E1 109.993} C_DIS
LIN {X 0.140,Y -597.278,Z 1425.409,A 0.000,B 0.000,C 90.000,E1 109.523} C_DIS
LIN {X -0.094,Y -602.055,Z 1425.406,A 0.000,B 0.000,C 90.000,E1 109.087} C_DIS
LIN {X 0.325,Y -608.086,Z 1425.403,A 0.000,B 0.000,C 90.000,E1 108.417} C_DIS
LIN {X -0.123,Y -613.276,Z 1425.399,A 0.000,B 0.000,C 90.000,E1 107.819} C_DIS
LIN {X 0.153,Y -616.862,Z 1425.396,A 0.000,B 0.000,C 90.000,E1 107.275} C_DIS
LIN {X -0.318,Y -620.064,Z 1425.393,A 0.000,B 0.000,C 90.000,E1 106.804} C_DIS
LIN {X 0.227,Y -621.385,Z 1425.392,A 0.000,B 0.000,C 90.000,E1 106.496} C_DIS
LIN {X -0.216,Y -623.473,Z 1425.389,A 0.000,B 0.000,C 90.000,E1 106.024} C_DIS
LIN {X 0.124,Y -625.105,Z 1425.386,A 0.000,B 0.000,C 90.000,E1 105.481} C_DIS
LIN {X -0.087,Y -625.690,Z 1425.385,A 0.000,B 0.000,C 90.000,E1 105.245} C_DIS
LIN {X -0.099,Y -626.969,Z 1425.380,A 0.000,B 0.000,C 90.000,E1 104.481} C_DIS
LIN {X 0.059,Y -628.084,Z 1425.376,A 0.000,B 0.000,C 90.000,E1 103.703} C_DIS
LIN {X 0.072,Y -628.928,Z 1425.372,A 0.000,B 0.000,C 90.000,E1 102.939} C_DIS
LIN {X -0.038,Y -629.220,Z 1425.368,A 0.000,B 0.000,C 90.000,E1 102.187} C_DIS
LIN {X 0.187,Y -629.140,Z 1425.365,A 0.000,B 0.000,C 90.000,E1 101.658} C_DIS
LIN {X -0.206,Y -628.715,Z 1425.362,A 0.000,B 0.000,C 90.000,E1 101.186} C_DIS
LIN {X 0.012,Y -628.043,Z 1425.359,A 0.000,B 0.000,C 90.000,E1 100.658} C_DIS
LIN {X -0.093,Y -626.567,Z 1425.355,A 0.000,B 0.000,C 90.000,E1 99.905} C_DIS
LIN {X 0.106,Y -625.309,Z 1425.352,A 0.000,B 0.000,C 90.000,E1 99.378} C_DIS
LIN {X 0.194,Y -623.790,Z 1425.349,A 0.000,B 0.000,C 90.000,E1 98.859} C_DIS
LIN {X -0.340,Y -621.984,Z 1425.347,A 0.000,B 0.000,C 90.000,E1 98.398} C_DIS
LIN {X -0.180,Y -619.758,Z 1425.344,A 0.000,B 0.000,C 90.000,E1 97.871} C_DIS
LIN {X 0.165,Y -616.021,Z 1425.339,A 0.000,B 0.000,C 90.000,E1 97.068} C_DIS
LIN {X 0.197,Y -613.371,Z 1425.337,A 0.000,B 0.000,C 90.000,E1 96.549} C_DIS
LIN {X 0.104,Y -609.418,Z 1425.333,A 0.000,B 0.000,C 90.000,E1 95.910} C_DIS
LIN {X 0.202,Y -607.020,Z 1425.331,A 0.000,B 0.000,C 90.000,E1 95.511} C_DIS
LIN {X -0.085,Y -605.049,Z 1425.329,A 0.000,B 0.000,C 90.000,E1 95.277} C_DIS
LIN {X 0.074,Y -601.818,Z 1425.327,A 0.000,B 0.000,C 90.000,E1 94.878} C_DIS
LIN {X 0.106,Y -596.905,Z 1425.324,A 0.000,B 0.000,C 90.000,E1 94.359} C_DIS
LIN {X 0.298,Y -591.416,Z 1425.322,A 0.000,B 0.000,C 90.000,E1 93.841} C_DIS
LIN {X 0.208,Y -585.525,Z 1425.319,A 0.000,B 0.000,C 90.000,E1 93.383} C_DIS
LIN {X 0.261,Y -582.496,Z 1425.318,A 0.000,B 0.000,C 90.000,E1 93.154} C_DIS
LIN {X 0.038,Y -577.585,Z 1425.316,A 0.000,B 0.000,C 90.000,E1 92.865} C_DIS
LIN {X 0.188,Y -573.127,Z 1425.314,A 0.000,B 0.000,C 90.000,E1 92.465} C_DIS
LIN {X 0.151,Y -573.101,Z 1425.314,A 0.000,B 0.000,C 90.000,E1 92.465} C_DIS
LIN {X 0.083,Y -572.318,Z 1425.313,A 0.000,B 0.000,C 90.000,E1 92.236} C_DIS
LIN {X 0.222,Y -571.933,Z 1425.311,A 0.000,B 0.000,C 90.000,E1 91.949} C_DIS
LIN {X -0.059,Y -571.920,Z 1425.308,A 0.000,B 0.000,C 90.000,E1 91.432} C_DIS
LIN {X -0.221,Y -572.461,Z 1425.303,A 0.000,B 0.000,C 90.000,E1 90.630} C_DIS
LIN {X 0.051,Y -573.921,Z 1425.294,A 0.000,B 0.000,C 90.000,E1 88.969} C_DIS
LIN {X -0.074,Y -574.722,Z 1425.290,A 0.000,B 0.000,C 90.000,E1 88.165} C_DIS
LIN {X 0.262,Y -576.227,Z 1425.281,A 0.000,B 0.000,C 90.000,E1 86.502} C_DIS
LIN {X -0.063,Y -577.538,Z 1425.273,A 0.000,B 0.000,C 90.000,E1 85.179} C_DIS
LIN {X -0.222,Y -579.129,Z 1425.264,A 0.000,B 0.000,C 90.000,E1 83.571} C_DIS
LIN {X -0.221,Y -580.923,Z 1425.255,A 0.000,B 0.000,C 90.000,E1 81.951} C_DIS
LIN {X 0.162,Y -582.364,Z 1425.248,A 0.000,B 0.000,C 90.000,E1 80.566} C_DIS
LIN {X -0.255,Y -584.085,Z 1425.239,A 0.000,B 0.000,C 90.000,E1 78.993} C_DIS
LIN {X -0.193,Y -585.481,Z 1425.231,A 0.000,B 0.000,C 90.000,E1 77.645} C_DIS
LIN {X -0.028,Y -586.142,Z 1425.227,A 0.000,B 0.000,C 90.000,E1 76.825} C_DIS
LIN {X 0.207,Y -587.126,Z 1425.219,A 0.000,B 0.000,C 90.000,E1 75.463} C_DIS
LIN {X 0.141,Y -588.198,Z 1425.210,A 0.000,B 0.000,C 90.000,E1 73.866} C_DIS
LIN {X 0.110,Y -589.236,Z 1425.200,A 0.000,B 0.000,C 90.000,E1 72.000} C_DIS
LIN {X 0.100,Y -590.238,Z 1425.190,A 0.000,B 0.000,C 90.000,E1 70.134} C_DIS
LIN {X 0.074,Y -591.140,Z 1425.181,A 0.000,B 0.000,C 90.000,E1 68.539} C_DIS
LIN {X 0.086,Y -592.486,Z 1425.169,A 0.000,B 0.000,C 90.000,E1 66.410} C_DIS
LIN {X 0.141,Y -593.844,Z 1425.157,A 0.000,B 0.000,C 90.000,E1 64.280} C_DIS
LIN {X 0.119,Y -595.153,Z 1425.148,A 0.000,B 0.000,C 90.000,E1 62.692} C_DIS
LIN {X -0.138,Y -596.428,Z 1425.140,A 0.000,B 0.000,C 90.000,E1 61.129} C_DIS
LIN {X -0.161,Y -598.018,Z 1425.129,A 0.000,B 0.000,C 90.000,E1 59.282} C_DIS
LIN {X -0.350,Y -599.779,Z 1425.119,A 0.000,B 0.000,C 90.000,E1 57.454} C_DIS
LIN {X -0.072,Y -601.178,Z 1425.110,A 0.000,B 0.000,C 90.000,E1 55.849} C_DIS
LIN {X 0.236,Y -602.137,Z 1425.104,A 0.000,B 0.000,C 90.000,E1 54.769} C_DIS
LIN {X 0.069,Y -603.409,Z 1425.096,A 0.000,B 0.000,C 90.000,E1 53.210} C_DIS
LIN {X 0.031,Y -604.377,Z 1425.088,A 0.000,B 0.000,C 90.000,E1 51.904} C_DIS
LIN {X 0.008,Y -605.281,Z 1425.081,A 0.000,B 0.000,C 90.000,E1 50.598} C_DIS
LIN {X -0.082,Y -605.876,Z 1425.074,A 0.000,B 0.000,C 90.000,E1 49.299} C_DIS
LIN {X 0.039,Y -606.070,Z 1425.068,A 0.000,B 0.000,C 90.000,E1 48.243} C_DIS
LIN {X 0.240,Y -606.319,Z 1425.057,A 0.000,B 0.000,C 90.000,E1 46.134} C_DIS
LIN {X 0.144,Y -606.241,Z 1425.049,A 0.000,B 0.000,C 90.000,E1 44.838} C_DIS
LIN {X -0.007,Y -606.037,Z 1425.045,A 0.000,B 0.000,C 90.000,E1 44.069} C_DIS
